LIN {X 0,Y 171.621,Z 603.214,A -85,B 0,C 180,E1 -26145.354,E2 -26145.354} C_VEL
LIN {X 0,Y 176.916,Z 615.978,A -85,B 0,C 180,E1 -26149,E2 -26149} C_VEL
LIN {X 0,Y 181.976,Z 626.134,A -85,B 0,C 180,E1 -26152.338,E2 -26152.338} C_VEL
LIN {X 0,Y 187.873,Z 635.706,A -85,B 0,C 180,E1 -26155.867,E2 -26155.867} C_VEL
LIN {X 0,Y 193.607,Z 643.258,A -85,B 0,C 180,E1 -26158.912,E2 -26158.912} C_VEL
LIN {X 0,Y 201.714,Z 651.879,A -85,B 0,C 180,E1 -26162.725,E2 -26162.725} C_VEL
LIN {X 0,Y 211.086,Z 659.54,A -85,B 0,C 180,E1 -26166.451,E2 -26166.451} C_VEL
LIN {X 0,Y 220.948,Z 665.783,A -85,B 0,C 180,E1 -26169.763,E2 -26169.763} C_VEL
LIN {X 0,Y 234.366,Z 672.498,A -85,B 0,C 180,E1 -26173.645,E2 -26173.645} C_VEL
LIN {X 0,Y 246.298,Z 677.555,A -85,B 0,C 180,E1 -26176.805,E2 -26176.805} C_VEL
LIN {X 0,Y 253.834,Z 680.558,A -85,B 0,C 180,E1 -26178.825,E2 -26178.825} C_VEL
LIN {X 0,Y 260.206,Z 683.111,A -85,B 0,C 180,E1 -26180.674,E2 -26180.674} C_VEL
LIN {X 0,Y 265.463,Z 685.211,A -85,B 0,C 180,E1 -26182.393,E2 -26182.393} C_VEL
LIN {X 0,Y 269.417,Z 686.886,A -85,B 0,C 180,E1 -26184.011,E2 -26184.011} C_VEL
LIN {X 0,Y 272.304,Z 688.198,A -85,B 0,C 180,E1 -26185.559,E2 -26185.559} C_VEL
LIN {X 0,Y 274.956,Z 689.105,A -85,B 0,C 180,E1 -26187.07,E2 -26187.07} C_VEL
LIN {X 0,Y 276.564,Z 689.664,A -85,B 0,C 180,E1 -26188.544,E2 -26188.544} C_VEL
LIN {X 0,Y 277.483,Z 689.842,A -85,B 0,C 180,E1 -26190,E2 -26190} C_VEL
LIN {X 0,Y 276.566,Z 689.663,A -85,B 0,C 180,E1 -26191.456,E2 -26191.456} C_VEL
LIN {X 0,Y 274.501,Z 688.974,A -85,B 0,C 180,E1 -26193.184,E2 -26193.184} C_VEL
LIN {X 0,Y 272.278,Z 688.199,A -85,B 0,C 180,E1 -26194.441,E2 -26194.441} C_VEL
LIN {X 0,Y 268.678,Z 686.595,A -85,B 0,C 180,E1 -26196.311,E2 -26196.311} C_VEL
LIN {X 0,Y 265.415,Z 685.213,A -85,B 0,C 180,E1 -26197.608,E2 -26197.608} C_VEL
LIN {X 0,Y 260.173,Z 683.112,A -85,B 0,C 180,E1 -26199.327,E2 -26199.327} C_VEL
LIN {X 0,Y 253.886,Z 680.557,A -85,B 0,C 180,E1 -26201.173,E2 -26201.173} C_VEL
LIN {X 0,Y 245.609,Z 677.259,A -85,B 0,C 180,E1 -26203.385,E2 -26203.385} C_VEL
LIN {X 0,Y 234.359,Z 672.513,A -85,B 0,C 180,E1 -26206.349,E2 -26206.349} C_VEL
LIN {X 0,Y 220.948,Z 665.784,A -85,B 0,C 180,E1 -26210.237,E2 -26210.237} C_VEL
LIN {X 0,Y 211.166,Z 659.537,A -85,B 0,C 180,E1 -26213.539,E2 -26213.539} C_VEL
LIN {X 0,Y 201.751,Z 651.903,A -85,B 0,C 180,E1 -26217.262,E2 -26217.262} C_VEL
LIN {X 0,Y 192.273,Z 641.586,A -85,B 0,C 180,E1 -26221.782,E2 -26221.782} C_VEL
LIN {X 0,Y 185.61,Z 632.244,A -85,B 0,C 180,E1 -26225.461,E2 -26225.461} C_VEL
LIN {X 0,Y 180.259,Z 622.941,A -85,B 0,C 180,E1 -26228.767,E2 -26228.767} C_VEL
LIN {X 0,Y 175.258,Z 612.247,A -85,B 0,C 180,E1 -26232.116,E2 -26232.116} C_VEL
LIN {X 0,Y 170.985,Z 601.587,A -85,B 0,C 180,E1 -26235.058,E2 -26235.058} C_VEL
LIN {X 0,Y 167.177,Z 590.937,A -85,B 0,C 180,E1 -26237.634,E2 -26237.634} C_VEL
LIN {X 0,Y 160.92,Z 572.907,A -85,B 0,C 180,E1 -26241.531,E2 -26241.531} C_VEL
LIN {X 0,Y 157.524,Z 564.607,A -85,B 0,C 180,E1 -26243.75,E2 -26243.75} C_VEL
LIN {X 0,Y 153.292,Z 555.729,A -85,B 0,C 180,E1 -26246.722,E2 -26246.722} C_VEL
LIN {X 0,Y 148.61,Z 547.106,A -85,B 0,C 180,E1 -26250.427,E2 -26250.427} C_VEL
LIN {X 0,Y 144.239,Z 539.962,A -85,B 0,C 180,E1 -26254.48,E2 -26254.48} C_VEL
LIN {X 0,Y 141.462,Z 535.851,A -85,B 0,C 180,E1 -26257.504,E2 -26257.504} C_VEL
LIN {X 0,Y 138.867,Z 531.989,A -85,B 0,C 180,E1 -26260.874,E2 -26260.874} C_VEL
LIN {X 0,Y 136.38,Z 528.521,A -85,B 0,C 180,E1 -26264.882,E2 -26264.882} C_VEL
LIN {X 0,Y 135.759,Z 527.362,A -85,B 0,C 180,E1 -26266.152,E2 -26266.152} C_VEL
LIN {X 0,Y 133.331,Z 524.419,A -85,B 0,C 180,E1 -26272.623,E2 -26272.623} C_VEL
LIN {X 0,Y 132.769,Z 522.602,A -85,B 0,C 180,E1 -26276.211,E2 -26276.211} C_VEL
LIN {X 0,Y 132.584,Z 521.985,A -85,B 0,C 180,E1 -26280.005,E2 -26280.005} C_VEL
LIN {X 0,Y 132.854,Z 522.928,A -85,B 0,C 180,E1 -26284.176,E2 -26284.176} C_VEL
LIN {X 0,Y 135.306,Z 527.03,A -85,B 0,C 180,E1 -26292.567,E2 -26292.567} C_VEL
LIN {X 0,Y 136.125,Z 527.942,A -85,B 0,C 180,E1 -26294.2,E2 -26294.2} C_VEL
LIN {X 0,Y 138.548,Z 531.658,A -85,B 0,C 180,E1 -26298.297,E2 -26298.297} C_VEL
LIN {X 0,Y 139.546,Z 533.014,A -85,B 0,C 180,E1 -26299.687,E2 -26299.687} C_VEL
LIN {X 0,Y 142.466,Z 537.271,A -85,B 0,C 180,E1 -26303.248,E2 -26303.248} C_VEL
LIN {X 0,Y 145.553,Z 542.106,A -85,B 0,C 180,E1 -26306.436,E2 -26306.436} C_VEL
LIN {X 0,Y 147.873,Z 546.115,A -85,B 0,C 180,E1 -26308.575,E2 -26308.575} C_VEL
LIN {X 0,Y 151.392,Z 554.209,A -85,B 0,C 180,E1 -26311.634,E2 -26311.634} C_VEL
LIN {X 0,Y 155.275,Z 564.625,A -85,B 0,C 180,E1 -26314.706,E2 -26314.706} C_VEL
LIN {X 0,Y 156.576,Z 568.776,A -85,B 0,C 180,E1 -26315.702,E2 -26315.702} C_VEL
LIN {X 0,Y 154.221,Z 595.964,A -85,B 0,C 180,E1 -26316.734,E2 -26316.734} C_VEL
LIN {X 0,Y 152.545,Z 606.818,A -85,B 0,C 180,E1 -26317.392,E2 -26317.392} C_VEL
LIN {X 0,Y 150.304,Z 616.608,A -85,B 0,C 180,E1 -26318.175,E2 -26318.175} C_VEL
LIN {X 0,Y 147.443,Z 626.404,A -85,B 0,C 180,E1 -26319.235,E2 -26319.235} C_VEL
LIN {X 0,Y 144.352,Z 635.168,A -85,B 0,C 180,E1 -26320.473,E2 -26320.473} C_VEL
LIN {X 0,Y 140.704,Z 643.886,A -85,B 0,C 180,E1 -26322.014,E2 -26322.014} C_VEL
LIN {X 0,Y 136.653,Z 652.394,A -85,B 0,C 180,E1 -26323.945,E2 -26323.945} C_VEL
LIN {X 0,Y 132.202,Z 660.561,A -85,B 0,C 180,E1 -26326.284,E2 -26326.284} C_VEL
LIN {X 0,Y 128.058,Z 667.504,A -85,B 0,C 180,E1 -26328.809,E2 -26328.809} C_VEL
LIN {X 0,Y 124.167,Z 673.491,A -85,B 0,C 180,E1 -26331.493,E2 -26331.493} C_VEL
LIN {X 0,Y 119.57,Z 680.174,A -85,B 0,C 180,E1 -26335.382,E2 -26335.382} C_VEL
LIN {X 0,Y 116.001,Z 685.08,A -85,B 0,C 180,E1 -26339.004,E2 -26339.004} C_VEL
LIN {X 0,Y 111.98,Z 690.174,A -85,B 0,C 180,E1 -26343.939,E2 -26343.939} C_VEL
LIN {X 0,Y 108.812,Z 694.141,A -85,B 0,C 180,E1 -26349.192,E2 -26349.192} C_VEL
LIN {X 0,Y 106.71,Z 697.085,A -85,B 0,C 180,E1 -26354.726,E2 -26354.726} C_VEL
LIN {X 0,Y 105.784,Z 698.592,A -85,B 0,C 180,E1 -26358.503,E2 -26358.503} C_VEL
LIN {X 0,Y 105.043,Z 700.131,A -85,B 0,C 180,E1 -26366.164,E2 -26366.164} C_VEL
LIN {X 0,Y 105.176,Z 700.418,A -85,B 0,C 180,E1 -26370,E2 -26370} C_VEL
LIN {X 0,Y 105.231,Z 699.528,A -85,B 0,C 180,E1 -26377.676,E2 -26377.676} C_VEL
LIN {X 0,Y 105.787,Z 698.592,A -85,B 0,C 180,E1 -26381.496,E2 -26381.496} C_VEL
LIN {X 0,Y 107.993,Z 695.232,A -85,B 0,C 180,E1 -26388.989,E2 -26388.989} C_VEL
LIN {X 0,Y 110.82,Z 691.602,A -85,B 0,C 180,E1 -26394.344,E2 -26394.344} C_VEL
LIN {X 0,Y 114.515,Z 686.868,A -85,B 0,C 180,E1 -26399.404,E2 -26399.404} C_VEL
LIN {X 0,Y 118.575,Z 681.494,A -85,B 0,C 180,E1 -26403.708,E2 -26403.708} C_VEL
LIN {X 0,Y 122.393,Z 676.116,A -85,B 0,C 180,E1 -26407.079,E2 -26407.079} C_VEL
LIN {X 0,Y 126.09,Z 670.624,A -85,B 0,C 180,E1 -26409.865,E2 -26409.865} C_VEL
LIN {X 0,Y 131.154,Z 662.411,A -85,B 0,C 180,E1 -26413.095,E2 -26413.095} C_VEL
LIN {X 0,Y 135.524,Z 654.59,A -85,B 0,C 180,E1 -26415.483,E2 -26415.483} C_VEL
LIN {X 0,Y 139.562,Z 646.512,A -85,B 0,C 180,E1 -26417.432,E2 -26417.432} C_VEL
LIN {X 0,Y 143.733,Z 636.756,A -85,B 0,C 180,E1 -26419.278,E2 -26419.278} C_VEL
LIN {X 0,Y 146.784,Z 628.37,A -85,B 0,C 180,E1 -26420.539,E2 -26420.539} C_VEL
LIN {X 0,Y 149.931,Z 617.868,A -85,B 0,C 180,E1 -26421.734,E2 -26421.734} C_VEL
LIN {X 0,Y 152.26,Z 608.189,A -85,B 0,C 180,E1 -26422.532,E2 -26422.532} C_VEL
LIN {X 0,Y 154.059,Z 597.555,A -85,B 0,C 180,E1 -26423.167,E2 -26423.167} C_VEL
LIN {X 0,Y 155.953,Z 576.912,A -85,B 0,C 180,E1 -26423.989,E2 -26423.989} C_VEL
LIN {X 0,Y 156.52,Z 568.606,A -85,B 0,C 180,E1 -26424.339,E2 -26424.339} C_VEL
LIN {X 0,Y 153.874,Z 560.714,A -85,B 0,C 180,E1 -26426.368,E2 -26426.368} C_VEL
LIN {X 0,Y 149.72,Z 550.16,A -85,B 0,C 180,E1 -26429.786,E2 -26429.786} C_VEL
LIN {X 0,Y 147.011,Z 544.436,A -85,B 0,C 180,E1 -26432.214,E2 -26432.214} C_VEL
LIN {X 0,Y 143.831,Z 539.389,A -85,B 0,C 180,E1 -26435.281,E2 -26435.281} C_VEL
LIN {X 0,Y 142.084,Z 536.551,A -85,B 0,C 180,E1 -26437.2,E2 -26437.2} C_VEL
LIN {X 0,Y 140.892,Z 535.032,A -85,B 0,C 180,E1 -26438.576,E2 -26438.576} C_VEL
LIN {X 0,Y 138.995,Z 533.903,A -85,B 0,C 180,E1 -26440.815,E2 -26440.815} C_VEL
LIN {X 0,Y 133.719,Z 533.482,A -85,B 0,C 180,E1 -26448.992,E2 -26448.992} C_VEL
LIN {X 0,Y 133.382,Z 533.176,A -85,B 0,C 180,E1 -26449.838,E2 -26449.838} C_VEL
LIN {X 0,Y 131.799,Z 529.387,A -85,B 0,C 180,E1 -26457.703,E2 -26457.703} C_VEL
LIN {X 0,Y 131.717,Z 529.047,A -85,B 0,C 180,E1 -26459.995,E2 -26459.995} C_VEL
LIN {X 0,Y 131.926,Z 529.956,A -85,B 0,C 180,E1 -26464.196,E2 -26464.196} C_VEL
LIN {X 0,Y 134.158,Z 533.971,A -85,B 0,C 180,E1 -26472.428,E2 -26472.428} C_VEL
LIN {X 0,Y 134.782,Z 534.696,A -85,B 0,C 180,E1 -26473.758,E2 -26473.758} C_VEL
LIN {X 0,Y 137.254,Z 538.568,A -85,B 0,C 180,E1 -26478.18,E2 -26478.18} C_VEL
LIN {X 0,Y 140.569,Z 543.731,A -85,B 0,C 180,E1 -26482.647,E2 -26482.647} C_VEL
LIN {X 0,Y 143.405,Z 548.348,A -85,B 0,C 180,E1 -26485.777,E2 -26485.777} C_VEL
LIN {X 0,Y 147.758,Z 556.106,A -85,B 0,C 180,E1 -26489.858,E2 -26489.858} C_VEL
LIN {X 0,Y 152.402,Z 565.552,A -85,B 0,C 180,E1 -26493.594,E2 -26493.594} C_VEL
LIN {X 0,Y 156.256,Z 574.926,A -85,B 0,C 180,E1 -26496.401,E2 -26496.401} C_VEL
LIN {X 0,Y 160.04,Z 586.179,A -85,B 0,C 180,E1 -26499.036,E2 -26499.036} C_VEL
LIN {X 0,Y 163.433,Z 597.185,A -85,B 0,C 180,E1 -26501.588,E2 -26501.588} C_VEL
LIN {X 0,Y 166.658,Z 607.047,A -85,B 0,C 180,E1 -26504.202,E2 -26504.202} C_VEL
LIN {X 0,Y 170.411,Z 617.155,A -85,B 0,C 180,E1 -26507.266,E2 -26507.266} C_VEL
LIN {X 0,Y 174.824,Z 627.17,A -85,B 0,C 180,E1 -26510.695,E2 -26510.695} C_VEL
LIN {X 0,Y 179.681,Z 635.973,A -85,B 0,C 180,E1 -26514.077,E2 -26514.077} C_VEL
LIN {X 0,Y 184.854,Z 643.572,A -85,B 0,C 180,E1 -26517.273,E2 -26517.273} C_VEL
LIN {X 0,Y 192.277,Z 652.277,A -85,B 0,C 180,E1 -26521.302,E2 -26521.302} C_VEL
LIN {X 0,Y 200.736,Z 659.845,A -85,B 0,C 180,E1 -26525.157,E2 -26525.157} C_VEL
LIN {X 0,Y 210.803,Z 666.663,A -85,B 0,C 180,E1 -26528.976,E2 -26528.976} C_VEL
LIN {X 0,Y 221.28,Z 672.126,A -85,B 0,C 180,E1 -26532.318,E2 -26532.318} C_VEL
LIN {X 0,Y 235.082,Z 677.867,A -85,B 0,C 180,E1 -26536.163,E2 -26536.163} C_VEL
LIN {X 0,Y 246.752,Z 682.108,A -85,B 0,C 180,E1 -26539.288,E2 -26539.288} C_VEL
LIN {X 0,Y 255.57,Z 685.165,A -85,B 0,C 180,E1 -26541.858,E2 -26541.858} C_VEL
LIN {X 0,Y 261.463,Z 687.257,A -85,B 0,C 180,E1 -26543.981,E2 -26543.981} C_VEL
LIN {X 0,Y 264.432,Z 688.418,A -85,B 0,C 180,E1 -26545.427,E2 -26545.427} C_VEL
LIN {X 0,Y 267.399,Z 689.359,A -85,B 0,C 180,E1 -26547.069,E2 -26547.069} C_VEL
LIN {X 0,Y 269.242,Z 689.867,A -85,B 0,C 180,E1 -26548.504,E2 -26548.504} C_VEL
LIN {X 0,Y 270.315,Z 690.041,A -85,B 0,C 180,E1 -26550,E2 -26550} C_VEL
LIN {X 0,Y 269.24,Z 689.867,A -85,B 0,C 180,E1 -26551.496,E2 -26551.496} C_VEL
LIN {X 0,Y 267.239,Z 689.317,A -85,B 0,C 180,E1 -26553.015,E2 -26553.015} C_VEL
LIN {X 0,Y 264.41,Z 688.418,A -85,B 0,C 180,E1 -26554.574,E2 -26554.574} C_VEL
LIN {X 0,Y 261.016,Z 687.117,A -85,B 0,C 180,E1 -26556.183,E2 -26556.183} C_VEL
LIN {X 0,Y 255.564,Z 685.178,A -85,B 0,C 180,E1 -26558.132,E2 -26558.132} C_VEL
LIN {X 0,Y 249.679,Z 683.135,A -85,B 0,C 180,E1 -26559.893,E2 -26559.893} C_VEL
LIN {X 0,Y 243.252,Z 680.857,A -85,B 0,C 180,E1 -26561.668,E2 -26561.668} C_VEL
LIN {X 0,Y 232.346,Z 676.846,A -85,B 0,C 180,E1 -26564.562,E2 -26564.562} C_VEL
LIN {X 0,Y 217.434,Z 670.286,A -85,B 0,C 180,E1 -26568.858,E2 -26568.858} C_VEL
LIN {X 0,Y 205.884,Z 663.53,A -85,B 0,C 180,E1 -26572.839,E2 -26572.839} C_VEL
LIN {X 0,Y 195.479,Z 655.394,A -85,B 0,C 180,E1 -26577.158,E2 -26577.158} C_VEL
LIN {X 0,Y 188.213,Z 647.777,A -85,B 0,C 180,E1 -26580.821,E2 -26580.821} C_VEL
LIN {X 0,Y 181.58,Z 639.028,A -85,B 0,C 180,E1 -26584.674,E2 -26584.674} C_VEL
LIN {X 0,Y 176.615,Z 630.661,A -85,B 0,C 180,E1 -26588.007,E2 -26588.007} C_VEL
LIN {X 0,Y 172.513,Z 622.049,A -85,B 0,C 180,E1 -26591.095,E2 -26591.095} C_VEL
LIN {X 0,Y 168.754,Z 612.855,A -85,B 0,C 180,E1 -26594.083,E2 -26594.083} C_VEL
LIN {X 0,Y 164.892,Z 601.852,A -85,B 0,C 180,E1 -26597.218,E2 -26597.218} C_VEL
LIN {X 0,Y 161.241,Z 590.184,A -85,B 0,C 180,E1 -26600.098,E2 -26600.098} C_VEL
LIN {X 0,Y 156.857,Z 576.56,A -85,B 0,C 180,E1 -26603.178,E2 -26603.178} C_VEL
LIN {X 0,Y 152.863,Z 566.622,A -85,B 0,C 180,E1 -26606.056,E2 -26606.056} C_VEL
LIN {X 0,Y 148.504,Z 557.612,A -85,B 0,C 180,E1 -26609.499,E2 -26609.499} C_VEL
LIN {X 0,Y 144.243,Z 549.708,A -85,B 0,C 180,E1 -26613.387,E2 -26613.387} C_VEL
LIN {X 0,Y 141.473,Z 545.217,A -85,B 0,C 180,E1 -26616.297,E2 -26616.297} C_VEL
LIN {X 0,Y 139.46,Z 542.029,A -85,B 0,C 180,E1 -26618.719,E2 -26618.719} C_VEL
LIN {X 0,Y 137.255,Z 538.56,A -85,B 0,C 180,E1 -26621.819,E2 -26621.819} C_VEL
LIN {X 0,Y 134.781,Z 534.7,A -85,B 0,C 180,E1 -26626.242,E2 -26626.242} C_VEL
LIN {X 0,Y 134.159,Z 533.961,A -85,B 0,C 180,E1 -26627.572,E2 -26627.572} C_VEL
LIN {X 0,Y 131.822,Z 529.519,A -85,B 0,C 180,E1 -26636.949,E2 -26636.949} C_VEL
LIN {X 0,Y 131.718,Z 529.04,A -85,B 0,C 180,E1 -26640.005,E2 -26640.005} C_VEL
LIN {X 0,Y 131.94,Z 529.991,A -85,B 0,C 180,E1 -26643.918,E2 -26643.918} C_VEL
LIN {X 0,Y 134.319,Z 534.061,A -85,B 0,C 180,E1 -26652.373,E2 -26652.373} C_VEL
LIN {X 0,Y 134.87,Z 534.887,A -85,B 0,C 180,E1 -26653.566,E2 -26653.566} C_VEL
LIN {X 0,Y 137.881,Z 539.509,A -85,B 0,C 180,E1 -26658.726,E2 -26658.726} C_VEL
LIN {X 0,Y 140.659,Z 543.824,A -85,B 0,C 180,E1 -26662.359,E2 -26662.359} C_VEL
LIN {X 0,Y 144.231,Z 549.666,A -85,B 0,C 180,E1 -26666.21,E2 -26666.21} C_VEL
LIN {X 0,Y 146.772,Z 555.356,A -85,B 0,C 180,E1 -26668.712,E2 -26668.712} C_VEL
LIN {X 0,Y 150.791,Z 566.153,A -85,B 0,C 180,E1 -26672.316,E2 -26672.316} C_VEL
LIN {X 0,Y 152.326,Z 571.077,A -85,B 0,C 180,E1 -26673.622,E2 -26673.622} C_VEL
LIN {X 0,Y 150.034,Z 596.193,A -85,B 0,C 180,E1 -26674.584,E2 -26674.584} C_VEL
LIN {X 0,Y 148.095,Z 608.002,A -85,B 0,C 180,E1 -26675.314,E2 -26675.314} C_VEL
LIN {X 0,Y 144.712,Z 621.282,A -85,B 0,C 180,E1 -26676.452,E2 -26676.452} C_VEL
LIN {X 0,Y 140.507,Z 633.383,A -85,B 0,C 180,E1 -26678.021,E2 -26678.021} C_VEL
LIN {X 0,Y 136.691,Z 642.379,A -85,B 0,C 180,E1 -26679.536,E2 -26679.536} C_VEL
LIN {X 0,Y 132.434,Z 651.101,A -85,B 0,C 180,E1 -26681.446,E2 -26681.446} C_VEL
LIN {X 0,Y 128.308,Z 658.516,A -85,B 0,C 180,E1 -26683.469,E2 -26683.469} C_VEL
LIN {X 0,Y 122.797,Z 667.308,A -85,B 0,C 180,E1 -26686.624,E2 -26686.624} C_VEL
LIN {X 0,Y 118.669,Z 673.294,A -85,B 0,C 180,E1 -26689.349,E2 -26689.349} C_VEL
LIN {X 0,Y 114.952,Z 678.499,A -85,B 0,C 180,E1 -26692.311,E2 -26692.311} C_VEL
LIN {X 0,Y 109.964,Z 684.884,A -85,B 0,C 180,E1 -26697.095,E2 -26697.095} C_VEL
LIN {X 0,Y 105.619,Z 689.977,A -85,B 0,C 180,E1 -26702.239,E2 -26702.239} C_VEL
LIN {X 0,Y 102.189,Z 693.944,A -85,B 0,C 180,E1 -26707.774,E2 -26707.774} C_VEL
LIN {X 0,Y 99.835,Z 696.887,A -85,B 0,C 180,E1 -26713.645,E2 -26713.645} C_VEL
LIN {X 0,Y 98.804,Z 698.395,A -85,B 0,C 180,E1 -26717.679,E2 -26717.679} C_VEL
LIN {X 0,Y 97.949,Z 699.935,A -85,B 0,C 180,E1 -26725.885,E2 -26725.885} C_VEL
LIN {X 0,Y 98.083,Z 700.222,A -85,B 0,C 180,E1 -26730,E2 -26730} C_VEL
LIN {X 0,Y 98.188,Z 699.331,A -85,B 0,C 180,E1 -26738.23,E2 -26738.23} C_VEL
LIN {X 0,Y 98.806,Z 698.395,A -85,B 0,C 180,E1 -26742.321,E2 -26742.321} C_VEL
LIN {X 0,Y 101.264,Z 695.034,A -85,B 0,C 180,E1 -26750.305,E2 -26750.305} C_VEL
LIN {X 0,Y 104.361,Z 691.405,A -85,B 0,C 180,E1 -26755.959,E2 -26755.959} C_VEL
LIN {X 0,Y 108.374,Z 686.672,A -85,B 0,C 180,E1 -26761.251,E2 -26761.251} C_VEL
LIN {X 0,Y 113.448,Z 680.404,A -85,B 0,C 180,E1 -26766.349,E2 -26766.349} C_VEL
LIN {X 0,Y 118.688,Z 673.295,A -85,B 0,C 180,E1 -26770.643,E2 -26770.643} C_VEL
LIN {X 0,Y 124.948,Z 664.064,A -85,B 0,C 180,E1 -26774.675,E2 -26774.675} C_VEL
LIN {X 0,Y 130.628,Z 654.393,A -85,B 0,C 180,E1 -26777.712,E2 -26777.712} C_VEL
LIN {X 0,Y 134.865,Z 646.316,A -85,B 0,C 180,E1 -26779.651,E2 -26779.651} C_VEL
LIN {X 0,Y 139.205,Z 636.56,A -85,B 0,C 180,E1 -26781.493,E2 -26781.493} C_VEL
LIN {X 0,Y 142.377,Z 628.174,A -85,B 0,C 180,E1 -26782.745,E2 -26782.745} C_VEL
LIN {X 0,Y 145.646,Z 617.672,A -85,B 0,C 180,E1 -26783.925,E2 -26783.925} C_VEL
LIN {X 0,Y 148.205,Z 607.314,A -85,B 0,C 180,E1 -26784.743,E2 -26784.743} C_VEL
LIN {X 0,Y 149.975,Z 596.932,A -85,B 0,C 180,E1 -26785.351,E2 -26785.351} C_VEL
LIN {X 0,Y 151.985,Z 575.616,A -85,B 0,C 180,E1 -26786.192,E2 -26786.192} C_VEL
LIN {X 0,Y 152.233,Z 570.793,A -85,B 0,C 180,E1 -26786.453,E2 -26786.453} C_VEL
LIN {X 0,Y 150.06,Z 564.182,A -85,B 0,C 180,E1 -26788.299,E2 -26788.299} C_VEL
LIN {X 0,Y 146.442,Z 554.498,A -85,B 0,C 180,E1 -26791.609,E2 -26791.609} C_VEL
LIN {X 0,Y 144.15,Z 549.512,A -85,B 0,C 180,E1 -26793.872,E2 -26793.872} C_VEL
LIN {X 0,Y 140.041,Z 542.737,A -85,B 0,C 180,E1 -26798.404,E2 -26798.404} C_VEL
LIN {X 0,Y 137.085,Z 538.343,A -85,B 0,C 180,E1 -26802.466,E2 -26802.466} C_VEL
LIN {X 0,Y 134.697,Z 534.461,A -85,B 0,C 180,E1 -26806.834,E2 -26806.834} C_VEL
LIN {X 0,Y 133.382,Z 533.176,A -85,B 0,C 180,E1 -26809.838,E2 -26809.838} C_VEL
LIN {X 0,Y 132.512,Z 532.627,A -85,B 0,C 180,E1 -26812.365,E2 -26812.365} C_VEL
LIN {X 0,Y 131.792,Z 532.955,A -85,B 0,C 180,E1 -26814.933,E2 -26814.933} C_VEL
LIN {X 0,Y 130.969,Z 535.132,A -85,B 0,C 180,E1 -26820.102,E2 -26820.102} C_VEL
LIN {X 0,Y 130.986,Z 536.834,A -85,B 0,C 180,E1 -26823.563,E2 -26823.563} C_VEL
LIN {X 0,Y 133.157,Z 540.966,A -85,B 0,C 180,E1 -26832.183,E2 -26832.183} C_VEL
LIN {X 0,Y 136.274,Z 546.089,A -85,B 0,C 180,E1 -26838.168,E2 -26838.168} C_VEL
LIN {X 0,Y 138.864,Z 550.396,A -85,B 0,C 180,E1 -26841.815,E2 -26841.815} C_VEL
LIN {X 0,Y 141.09,Z 554.185,A -85,B 0,C 180,E1 -26844.455,E2 -26844.455} C_VEL
LIN {X 0,Y 145.036,Z 561.671,A -85,B 0,C 180,E1 -26848.487,E2 -26848.487} C_VEL
LIN {X 0,Y 149.247,Z 570.719,A -85,B 0,C 180,E1 -26852.172,E2 -26852.172} C_VEL
LIN {X 0,Y 152.826,Z 579.943,A -85,B 0,C 180,E1 -26855.011,E2 -26855.011} C_VEL
LIN {X 0,Y 155.977,Z 590.349,A -85,B 0,C 180,E1 -26857.561,E2 -26857.561} C_VEL
LIN {X 0,Y 158.362,Z 599.183,A -85,B 0,C 180,E1 -26859.737,E2 -26859.737} C_VEL
LIN {X 0,Y 161.065,Z 608.7,A -85,B 0,C 180,E1 -26862.383,E2 -26862.383} C_VEL
LIN {X 0,Y 163.883,Z 617.554,A -85,B 0,C 180,E1 -26865.153,E2 -26865.153} C_VEL
LIN {X 0,Y 167.126,Z 626.218,A -85,B 0,C 180,E1 -26868.185,E2 -26868.185} C_VEL
LIN {X 0,Y 170.873,Z 634.482,A -85,B 0,C 180,E1 -26871.389,E2 -26871.389} C_VEL
LIN {X 0,Y 176.446,Z 644.006,A -85,B 0,C 180,E1 -26875.553,E2 -26875.553} C_VEL
LIN {X 0,Y 183.092,Z 652.655,A -85,B 0,C 180,E1 -26879.749,E2 -26879.749} C_VEL
LIN {X 0,Y 190.671,Z 660.146,A -85,B 0,C 180,E1 -26883.749,E2 -26883.749} C_VEL
LIN {X 0,Y 198.336,Z 665.908,A -85,B 0,C 180,E1 -26887.108,E2 -26887.108} C_VEL
LIN {X 0,Y 208.351,Z 671.711,A -85,B 0,C 180,E1 -26890.808,E2 -26890.808} C_VEL
LIN {X 0,Y 219.133,Z 676.52,A -85,B 0,C 180,E1 -26894.173,E2 -26894.173} C_VEL
LIN {X 0,Y 232.109,Z 681.172,A -85,B 0,C 180,E1 -26897.763,E2 -26897.763} C_VEL
LIN {X 0,Y 242.25,Z 684.363,A -85,B 0,C 180,E1 -26900.515,E2 -26900.515} C_VEL
LIN {X 0,Y 248.219,Z 686.173,A -85,B 0,C 180,E1 -26902.274,E2 -26902.274} C_VEL
LIN {X 0,Y 254.236,Z 687.958,A -85,B 0,C 180,E1 -26904.334,E2 -26904.334} C_VEL
LIN {X 0,Y 256.368,Z 688.643,A -85,B 0,C 180,E1 -26905.283,E2 -26905.283} C_VEL
LIN {X 0,Y 260.299,Z 689.748,A -85,B 0,C 180,E1 -26907.356,E2 -26907.356} C_VEL
LIN {X 0,Y 261.821,Z 690.072,A -85,B 0,C 180,E1 -26908.462,E2 -26908.462} C_VEL
LIN {X 0,Y 263.123,Z 690.239,A -85,B 0,C 180,E1 -26910,E2 -26910} C_VEL
LIN {X 0,Y 261.817,Z 690.071,A -85,B 0,C 180,E1 -26911.538,E2 -26911.538} C_VEL
LIN {X 0,Y 259.449,Z 689.531,A -85,B 0,C 180,E1 -26913.106,E2 -26913.106} C_VEL
LIN {X 0,Y 256.345,Z 688.643,A -85,B 0,C 180,E1 -26914.718,E2 -26914.718} C_VEL
LIN {X 0,Y 254.232,Z 687.965,A -85,B 0,C 180,E1 -26915.658,E2 -26915.658} C_VEL
LIN {X 0,Y 248.218,Z 686.176,A -85,B 0,C 180,E1 -26917.724,E2 -26917.724} C_VEL
LIN {X 0,Y 239.977,Z 683.679,A -85,B 0,C 180,E1 -26920.12,E2 -26920.12} C_VEL
LIN {X 0,Y 230.5,Z 680.631,A -85,B 0,C 180,E1 -26922.676,E2 -26922.676} C_VEL
LIN {X 0,Y 214.81,Z 674.704,A -85,B 0,C 180,E1 -26927.125,E2 -26927.125} C_VEL
LIN {X 0,Y 203.242,Z 668.921,A -85,B 0,C 180,E1 -26931,E2 -26931} C_VEL
LIN {X 0,Y 193.666,Z 662.535,A -85,B 0,C 180,E1 -26934.884,E2 -26934.884} C_VEL
LIN {X 0,Y 186.106,Z 655.804,A -85,B 0,C 180,E1 -26938.606,E2 -26938.606} C_VEL
LIN {X 0,Y 179.276,Z 647.971,A -85,B 0,C 180,E1 -26942.568,E2 -26942.568} C_VEL
LIN {X 0,Y 174.048,Z 640.217,A -85,B 0,C 180,E1 -26946.146,E2 -26946.146} C_VEL
LIN {X 0,Y 169.699,Z 632.112,A -85,B 0,C 180,E1 -26949.557,E2 -26949.557} C_VEL
LIN {X 0,Y 165.816,Z 622.857,A -85,B 0,C 180,E1 -26953.025,E2 -26953.025} C_VEL
LIN {X 0,Y 162.519,Z 613.253,A -85,B 0,C 180,E1 -26956.225,E2 -26956.225} C_VEL
LIN {X 0,Y 159.259,Z 602.507,A -85,B 0,C 180,E1 -26959.396,E2 -26959.396} C_VEL
LIN {X 0,Y 156.191,Z 591.08,A -85,B 0,C 180,E1 -26962.296,E2 -26962.296} C_VEL
LIN {X 0,Y 152.909,Z 580.112,A -85,B 0,C 180,E1 -26964.93,E2 -26964.93} C_VEL
LIN {X 0,Y 149.16,Z 570.549,A -85,B 0,C 180,E1 -26967.896,E2 -26967.896} C_VEL
LIN {X 0,Y 145.19,Z 562.04,A -85,B 0,C 180,E1 -26971.363,E2 -26971.363} C_VEL
LIN {X 0,Y 141.548,Z 554.977,A -85,B 0,C 180,E1 -26975.042,E2 -26975.042} C_VEL
LIN {X 0,Y 138.144,Z 549.065,A -85,B 0,C 180,E1 -26979.143,E2 -26979.143} C_VEL
LIN {X 0,Y 135.497,Z 544.882,A -85,B 0,C 180,E1 -26983.09,E2 -26983.09} C_VEL
LIN {X 0,Y 133.157,Z 540.966,A -85,B 0,C 180,E1 -26987.817,E2 -26987.817} C_VEL
LIN {X 0,Y 131.111,Z 537.419,A -85,B 0,C 180,E1 -26995.2,E2 -26995.2} C_VEL
LIN {X 0,Y 130.897,Z 536.44,A -85,B 0,C 180,E1 -26997.697,E2 -26997.697} C_VEL
LIN {X 0,Y 130.857,Z 536.195,A -85,B 0,C 180,E1 -27000.774,E2 -27000.774} C_VEL
LIN {X 0,Y 131.03,Z 537.046,A -85,B 0,C 180,E1 -27003.657,E2 -27003.657} C_VEL
LIN {X 0,Y 133.164,Z 540.952,A -85,B 0,C 180,E1 -27011.805,E2 -27011.805} C_VEL
LIN {X 0,Y 136.198,Z 545.92,A -85,B 0,C 180,E1 -27017.652,E2 -27017.652} C_VEL
LIN {X 0,Y 138.95,Z 550.524,A -85,B 0,C 180,E1 -27021.532,E2 -27021.532} C_VEL
LIN {X 0,Y 141.931,Z 555.68,A -85,B 0,C 180,E1 -27024.984,E2 -27024.984} C_VEL
LIN {X 0,Y 144.41,Z 561.744,A -85,B 0,C 180,E1 -27027.641,E2 -27027.641} C_VEL
LIN {X 0,Y 148.057,Z 572.635,A -85,B 0,C 180,E1 -27031.213,E2 -27031.213} C_VEL
LIN {X 0,Y 148.279,Z 573.652,A -85,B 0,C 180,E1 -27031.445,E2 -27031.445} C_VEL
LIN {X 0,Y 146.028,Z 596.711,A -85,B 0,C 180,E1 -27032.325,E2 -27032.325} C_VEL
LIN {X 0,Y 143.82,Z 609.218,A -85,B 0,C 180,E1 -27033.097,E2 -27033.097} C_VEL
LIN {X 0,Y 140.279,Z 622.078,A -85,B 0,C 180,E1 -27034.245,E2 -27034.245} C_VEL
LIN {X 0,Y 136.248,Z 633.187,A -85,B 0,C 180,E1 -27035.668,E2 -27035.668} C_VEL
LIN {X 0,Y 132.275,Z 642.182,A -85,B 0,C 180,E1 -27037.159,E2 -27037.159} C_VEL
LIN {X 0,Y 127.837,Z 650.904,A -85,B 0,C 180,E1 -27039.056,E2 -27039.056} C_VEL
LIN {X 0,Y 123.532,Z 658.32,A -85,B 0,C 180,E1 -27041.078,E2 -27041.078} C_VEL
LIN {X 0,Y 117.728,Z 667.111,A -85,B 0,C 180,E1 -27044.245,E2 -27044.245} C_VEL
LIN {X 0,Y 113.364,Z 673.098,A -85,B 0,C 180,E1 -27047.005,E2 -27047.005} C_VEL
LIN {X 0,Y 108.289,Z 679.596,A -85,B 0,C 180,E1 -27050.95,E2 -27050.95} C_VEL
LIN {X 0,Y 104.058,Z 684.687,A -85,B 0,C 180,E1 -27054.965,E2 -27054.965} C_VEL
LIN {X 0,Y 99.35,Z 689.779,A -85,B 0,C 180,E1 -27060.319,E2 -27060.319} C_VEL
LIN {X 0,Y 95.616,Z 693.746,A -85,B 0,C 180,E1 -27066.155,E2 -27066.155} C_VEL
LIN {X 0,Y 93.01,Z 696.69,A -85,B 0,C 180,E1 -27072.408,E2 -27072.408} C_VEL
LIN {X 0,Y 91.857,Z 698.198,A -85,B 0,C 180,E1 -27076.731,E2 -27076.731} C_VEL
LIN {X 0,Y 90.879,Z 699.739,A -85,B 0,C 180,E1 -27085.565,E2 -27085.565} C_VEL
LIN {X 0,Y 90.981,Z 700.026,A -85,B 0,C 180,E1 -27090,E2 -27090} C_VEL
LIN {X 0,Y 91.149,Z 699.134,A -85,B 0,C 180,E1 -27098.871,E2 -27098.871} C_VEL
LIN {X 0,Y 91.859,Z 698.198,A -85,B 0,C 180,E1 -27103.269,E2 -27103.269} C_VEL
LIN {X 0,Y 94.601,Z 694.837,A -85,B 0,C 180,E1 -27111.805,E2 -27111.805} C_VEL
LIN {X 0,Y 98.001,Z 691.208,A -85,B 0,C 180,E1 -27117.784,E2 -27117.784} C_VEL
LIN {X 0,Y 102.362,Z 686.475,A -85,B 0,C 180,E1 -27123.316,E2 -27123.316} C_VEL
LIN {X 0,Y 105.72,Z 682.688,A -85,B 0,C 180,E1 -27126.748,E2 -27126.748} C_VEL
LIN {X 0,Y 110.349,Z 677.033,A -85,B 0,C 180,E1 -27130.753,E2 -27130.753} C_VEL
LIN {X 0,Y 115.515,Z 670.231,A -85,B 0,C 180,E1 -27134.4,E2 -27134.4} C_VEL
LIN {X 0,Y 121.155,Z 662.018,A -85,B 0,C 180,E1 -27137.697,E2 -27137.697} C_VEL
LIN {X 0,Y 125.962,Z 654.197,A -85,B 0,C 180,E1 -27140.1,E2 -27140.1} C_VEL
LIN {X 0,Y 130.369,Z 646.119,A -85,B 0,C 180,E1 -27142.037,E2 -27142.037} C_VEL
LIN {X 0,Y 134.893,Z 636.364,A -85,B 0,C 180,E1 -27143.857,E2 -27143.857} C_VEL
LIN {X 0,Y 138.201,Z 627.978,A -85,B 0,C 180,E1 -27145.085,E2 -27145.085} C_VEL
LIN {X 0,Y 141.591,Z 617.476,A -85,B 0,C 180,E1 -27146.242,E2 -27146.242} C_VEL
LIN {X 0,Y 144.291,Z 606.704,A -85,B 0,C 180,E1 -27147.083,E2 -27147.083} C_VEL
LIN {X 0,Y 146.058,Z 596.62,A -85,B 0,C 180,E1 -27147.655,E2 -27147.655} C_VEL
LIN {X 0,Y 148.301,Z 573.653,A -85,B 0,C 180,E1 -27148.541,E2 -27148.541} C_VEL
LIN {X 0,Y 146.446,Z 567.698,A -85,B 0,C 180,E1 -27150.308,E2 -27150.308} C_VEL
LIN {X 0,Y 143.238,Z 558.686,A -85,B 0,C 180,E1 -27153.594,E2 -27153.594} C_VEL
LIN {X 0,Y 141.591,Z 555.062,A -85,B 0,C 180,E1 -27155.383,E2 -27155.383} C_VEL
LIN {X 0,Y 138.221,Z 549.136,A -85,B 0,C 180,E1 -27159.438,E2 -27159.438} C_VEL
LIN {X 0,Y 135.425,Z 544.757,A -85,B 0,C 180,E1 -27163.604,E2 -27163.604} C_VEL
LIN {X 0,Y 133.164,Z 540.956,A -85,B 0,C 180,E1 -27168.195,E2 -27168.195} C_VEL
LIN {X 0,Y 130.929,Z 536.476,A -85,B 0,C 180,E1 -27177.688,E2 -27177.688} C_VEL
LIN {X 0,Y 130.85,Z 536.104,A -85,B 0,C 180,E1 -27179.995,E2 -27179.995} C_VEL
LIN {X 0,Y 130.986,Z 536.834,A -85,B 0,C 180,E1 -27183.563,E2 -27183.563} C_VEL
LIN {X 0,Y 131.078,Z 538.295,A -85,B 0,C 180,E1 -27185.19,E2 -27185.19} C_VEL
LIN {X 0,Y 131.458,Z 546.478,A -85,B 0,C 180,E1 -27189.901,E2 -27189.901} C_VEL
LIN {X 0,Y 131.977,Z 547.819,A -85,B 0,C 180,E1 -27191.51,E2 -27191.51} C_VEL
LIN {X 0,Y 134.764,Z 552.764,A -85,B 0,C 180,E1 -27197.298,E2 -27197.298} C_VEL
LIN {X 0,Y 137.158,Z 557.016,A -85,B 0,C 180,E1 -27200.92,E2 -27200.92} C_VEL
LIN {X 0,Y 139.714,Z 561.676,A -85,B 0,C 180,E1 -27204.119,E2 -27204.119} C_VEL
LIN {X 0,Y 143.51,Z 569.641,A -85,B 0,C 180,E1 -27208.177,E2 -27208.177} C_VEL
LIN {X 0,Y 146.765,Z 577.39,A -85,B 0,C 180,E1 -27211.211,E2 -27211.211} C_VEL
LIN {X 0,Y 149.807,Z 586.034,A -85,B 0,C 180,E1 -27213.85,E2 -27213.85} C_VEL
LIN {X 0,Y 152.83,Z 598.455,A -85,B 0,C 180,E1 -27217.017,E2 -27217.017} C_VEL
LIN {X 0,Y 155.346,Z 609.108,A -85,B 0,C 180,E1 -27220.051,E2 -27220.051} C_VEL
LIN {X 0,Y 157.713,Z 618.028,A -85,B 0,C 180,E1 -27222.934,E2 -27222.934} C_VEL
LIN {X 0,Y 160.547,Z 627.138,A -85,B 0,C 180,E1 -27226.236,E2 -27226.236} C_VEL
LIN {X 0,Y 164.211,Z 636.496,A -85,B 0,C 180,E1 -27230.061,E2 -27230.061} C_VEL
LIN {X 0,Y 168.342,Z 644.366,A -85,B 0,C 180,E1 -27233.671,E2 -27233.671} C_VEL
LIN {X 0,Y 174.097,Z 652.807,A -85,B 0,C 180,E1 -27237.958,E2 -27237.958} C_VEL
LIN {X 0,Y 181.057,Z 660.437,A -85,B 0,C 180,E1 -27242.239,E2 -27242.239} C_VEL
LIN {X 0,Y 189.316,Z 667.107,A -85,B 0,C 180,E1 -27246.372,E2 -27246.372} C_VEL
LIN {X 0,Y 198.155,Z 672.483,A -85,B 0,C 180,E1 -27250.02,E2 -27250.02} C_VEL
LIN {X 0,Y 208.731,Z 677.329,A -85,B 0,C 180,E1 -27253.645,E2 -27253.645} C_VEL
LIN {X 0,Y 222.918,Z 682.217,A -85,B 0,C 180,E1 -27257.765,E2 -27257.765} C_VEL
LIN {X 0,Y 228.928,Z 683.991,A -85,B 0,C 180,E1 -27259.386,E2 -27259.386} C_VEL
LIN {X 0,Y 236.566,Z 686.005,A -85,B 0,C 180,E1 -27261.458,E2 -27261.458} C_VEL
LIN {X 0,Y 242.966,Z 687.615,A -85,B 0,C 180,E1 -27263.356,E2 -27263.356} C_VEL
LIN {X 0,Y 248.091,Z 688.874,A -85,B 0,C 180,E1 -27265.125,E2 -27265.125} C_VEL
LIN {X 0,Y 253.206,Z 690.072,A -85,B 0,C 180,E1 -27267.655,E2 -27267.655} C_VEL
LIN {X 0,Y 254.33,Z 690.277,A -85,B 0,C 180,E1 -27268.417,E2 -27268.417} C_VEL
LIN {X 0,Y 255.899,Z 690.439,A -85,B 0,C 180,E1 -27270,E2 -27270} C_VEL
LIN {X 0,Y 254.324,Z 690.277,A -85,B 0,C 180,E1 -27271.583,E2 -27271.583} C_VEL
LIN {X 0,Y 251.531,Z 689.748,A -85,B 0,C 180,E1 -27273.203,E2 -27273.203} C_VEL
LIN {X 0,Y 248.07,Z 688.874,A -85,B 0,C 180,E1 -27274.876,E2 -27274.876} C_VEL
LIN {X 0,Y 240.884,Z 687.129,A -85,B 0,C 180,E1 -27277.288,E2 -27277.288} C_VEL
LIN {X 0,Y 234.82,Z 685.533,A -85,B 0,C 180,E1 -27279.03,E2 -27279.03} C_VEL
LIN {X 0,Y 228.825,Z 683.946,A -85,B 0,C 180,E1 -27280.652,E2 -27280.652} C_VEL
LIN {X 0,Y 217.138,Z 680.417,A -85,B 0,C 180,E1 -27283.848,E2 -27283.848} C_VEL
LIN {X 0,Y 203.352,Z 675.034,A -85,B 0,C 180,E1 -27288.122,E2 -27288.122} C_VEL
LIN {X 0,Y 193.756,Z 669.986,A -85,B 0,C 180,E1 -27291.734,E2 -27291.734} C_VEL
LIN {X 0,Y 184.021,Z 663.092,A -85,B 0,C 180,E1 -27296.178,E2 -27296.178} C_VEL
LIN {X 0,Y 176.901,Z 656.128,A -85,B 0,C 180,E1 -27300.23,E2 -27300.23} C_VEL
LIN {X 0,Y 170.576,Z 648.064,A -85,B 0,C 180,E1 -27304.517,E2 -27304.517} C_VEL
LIN {X 0,Y 165.878,Z 639.955,A -85,B 0,C 180,E1 -27308.396,E2 -27308.396} C_VEL
LIN {X 0,Y 162.12,Z 631.327,A -85,B 0,C 180,E1 -27312.088,E2 -27312.088} C_VEL
LIN {X 0,Y 158.928,Z 622.166,A -85,B 0,C 180,E1 -27315.612,E2 -27315.612} C_VEL
LIN {X 0,Y 156.235,Z 612.579,A -85,B 0,C 180,E1 -27318.869,E2 -27318.869} C_VEL
LIN {X 0,Y 153.76,Z 602.382,A -85,B 0,C 180,E1 -27321.904,E2 -27321.904} C_VEL
LIN {X 0,Y 151.316,Z 591.592,A -85,B 0,C 180,E1 -27324.719,E2 -27324.719} C_VEL
LIN {X 0,Y 148.543,Z 582.164,A -85,B 0,C 180,E1 -27327.244,E2 -27327.244} C_VEL
LIN {X 0,Y 145.153,Z 573.427,A -85,B 0,C 180,E1 -27330.251,E2 -27330.251} C_VEL
LIN {X 0,Y 141.601,Z 565.559,A -85,B 0,C 180,E1 -27333.771,E2 -27333.771} C_VEL
LIN {X 0,Y 138.095,Z 558.582,A -85,B 0,C 180,E1 -27337.861,E2 -27337.861} C_VEL
LIN {X 0,Y 135.718,Z 554.473,A -85,B 0,C 180,E1 -27341.159,E2 -27341.159} C_VEL
LIN {X 0,Y 134.115,Z 551.634,A -85,B 0,C 180,E1 -27343.841,E2 -27343.841} C_VEL
LIN {X 0,Y 131.983,Z 547.826,A -85,B 0,C 180,E1 -27348.475,E2 -27348.475} C_VEL
LIN {X 0,Y 130.115,Z 544.039,A -85,B 0,C 180,E1 -27356.327,E2 -27356.327} C_VEL
LIN {X 0,Y 129.979,Z 543.251,A -85,B 0,C 180,E1 -27359.23,E2 -27359.23} C_VEL
LIN {X 0,Y 130.054,Z 543.611,A -85,B 0,C 180,E1 -27362.328,E2 -27362.328} C_VEL
LIN {X 0,Y 132.278,Z 548.331,A -85,B 0,C 180,E1 -27371.886,E2 -27371.886} C_VEL
LIN {X 0,Y 134.823,Z 552.841,A -85,B 0,C 180,E1 -27377.005,E2 -27377.005} C_VEL
LIN {X 0,Y 137.228,Z 557.096,A -85,B 0,C 180,E1 -27380.62,E2 -27380.62} C_VEL
LIN {X 0,Y 139.931,Z 562.171,A -85,B 0,C 180,E1 -27383.99,E2 -27383.99} C_VEL
LIN {X 0,Y 142.331,Z 569.087,A -85,B 0,C 180,E1 -27386.822,E2 -27386.822} C_VEL
LIN {X 0,Y 144.462,Z 575.847,A -85,B 0,C 180,E1 -27389.115,E2 -27389.115} C_VEL
LIN {X 0,Y 142.428,Z 596.022,A -85,B 0,C 180,E1 -27389.887,E2 -27389.887} C_VEL
LIN {X 0,Y 140.205,Z 608.393,A -85,B 0,C 180,E1 -27390.628,E2 -27390.628} C_VEL
LIN {X 0,Y 136.415,Z 621.882,A -85,B 0,C 180,E1 -27391.782,E2 -27391.782} C_VEL
LIN {X 0,Y 132.233,Z 632.991,A -85,B 0,C 180,E1 -27393.167,E2 -27393.167} C_VEL
LIN {X 0,Y 128.111,Z 641.986,A -85,B 0,C 180,E1 -27394.627,E2 -27394.627} C_VEL
LIN {X 0,Y 123.48,Z 650.708,A -85,B 0,C 180,E1 -27396.493,E2 -27396.493} C_VEL
LIN {X 0,Y 118.974,Z 658.123,A -85,B 0,C 180,E1 -27398.492,E2 -27398.492} C_VEL
LIN {X 0,Y 112.859,Z 666.914,A -85,B 0,C 180,E1 -27401.646,E2 -27401.646} C_VEL
LIN {X 0,Y 108.259,Z 672.901,A -85,B 0,C 180,E1 -27404.431,E2 -27404.431} C_VEL
LIN {X 0,Y 102.604,Z 679.656,A -85,B 0,C 180,E1 -27408.633,E2 -27408.633} C_VEL
LIN {X 0,Y 98.295,Z 684.489,A -85,B 0,C 180,E1 -27412.574,E2 -27412.574} C_VEL
LIN {X 0,Y 93.209,Z 689.582,A -85,B 0,C 180,E1 -27418.143,E2 -27418.143} C_VEL
LIN {X 0,Y 89.14,Z 693.549,A -85,B 0,C 180,E1 -27424.302,E2 -27424.302} C_VEL
LIN {X 0,Y 86.243,Z 696.493,A -85,B 0,C 180,E1 -27430.976,E2 -27430.976} C_VEL
LIN {X 0,Y 84.949,Z 698.001,A -85,B 0,C 180,E1 -27435.629,E2 -27435.629} C_VEL
LIN {X 0,Y 83.795,Z 699.542,A -85,B 0,C 180,E1 -27445.189,E2 -27445.189} C_VEL
LIN {X 0,Y 83.888,Z 699.83,A -85,B 0,C 180,E1 -27450,E2 -27450} C_VEL
LIN {X 0,Y 84.136,Z 698.938,A -85,B 0,C 180,E1 -27459.617,E2 -27459.617} C_VEL
LIN {X 0,Y 84.95,Z 698.001,A -85,B 0,C 180,E1 -27464.37,E2 -27464.37} C_VEL
LIN {X 0,Y 88.012,Z 694.64,A -85,B 0,C 180,E1 -27473.532,E2 -27473.532} C_VEL
LIN {X 0,Y 91.754,Z 691.011,A -85,B 0,C 180,E1 -27479.859,E2 -27479.859} C_VEL
LIN {X 0,Y 96.5,Z 686.279,A -85,B 0,C 180,E1 -27485.635,E2 -27485.635} C_VEL
LIN {X 0,Y 100.095,Z 682.491,A -85,B 0,C 180,E1 -27489.191,E2 -27489.191} C_VEL
LIN {X 0,Y 105.044,Z 676.836,A -85,B 0,C 180,E1 -27493.296,E2 -27493.296} C_VEL
LIN {X 0,Y 110.531,Z 670.034,A -85,B 0,C 180,E1 -27496.988,E2 -27496.988} C_VEL
LIN {X 0,Y 116.477,Z 661.821,A -85,B 0,C 180,E1 -27500.291,E2 -27500.291} C_VEL
LIN {X 0,Y 121.515,Z 654,A -85,B 0,C 180,E1 -27502.678,E2 -27502.678} C_VEL
LIN {X 0,Y 126.124,Z 645.923,A -85,B 0,C 180,E1 -27504.581,E2 -27504.581} C_VEL
LIN {X 0,Y 130.827,Z 636.167,A -85,B 0,C 180,E1 -27506.371,E2 -27506.371} C_VEL
LIN {X 0,Y 134.273,Z 627.782,A -85,B 0,C 180,E1 -27507.564,E2 -27507.564} C_VEL
LIN {X 0,Y 137.772,Z 617.28,A -85,B 0,C 180,E1 -27508.697,E2 -27508.697} C_VEL
LIN {X 0,Y 140.473,Z 606.952,A -85,B 0,C 180,E1 -27509.481,E2 -27509.481} C_VEL
LIN {X 0,Y 142.353,Z 596.698,A -85,B 0,C 180,E1 -27510.056,E2 -27510.056} C_VEL
LIN {X 0,Y 144.403,Z 577.013,A -85,B 0,C 180,E1 -27510.811,E2 -27510.811} C_VEL
LIN {X 0,Y 144.361,Z 575.543,A -85,B 0,C 180,E1 -27510.988,E2 -27510.988} C_VEL
LIN {X 0,Y 141.046,Z 565.171,A -85,B 0,C 180,E1 -27514.67,E2 -27514.67} C_VEL
LIN {X 0,Y 139.403,Z 561.062,A -85,B 0,C 180,E1 -27516.637,E2 -27516.637} C_VEL
LIN {X 0,Y 136.361,Z 555.416,A -85,B 0,C 180,E1 -27520.618,E2 -27520.618} C_VEL
LIN {X 0,Y 133.917,Z 551.33,A -85,B 0,C 180,E1 -27524.588,E2 -27524.588} C_VEL
LIN {X 0,Y 131.984,Z 547.805,A -85,B 0,C 180,E1 -27528.866,E2 -27528.866} C_VEL
LIN {X 0,Y 130.017,Z 543.376,A -85,B 0,C 180,E1 -27538.447,E2 -27538.447} C_VEL
LIN {X 0,Y 129.984,Z 543.161,A -85,B 0,C 180,E1 -27539.995,E2 -27539.995} C_VEL
LIN {X 0,Y 130.1,Z 543.949,A -85,B 0,C 180,E1 -27543.479,E2 -27543.479} C_VEL
LIN {X 0,Y 131.977,Z 547.819,A -85,B 0,C 180,E1 -27551.51,E2 -27551.51} C_VEL
LIN {X 0,Y 132.631,Z 548.898,A -85,B 0,C 180,E1 -27553.104,E2 -27553.104} C_VEL
LIN {X 0,Y 133.226,Z 550.73,A -85,B 0,C 180,E1 -27554.571,E2 -27554.571} C_VEL
LIN {X 0,Y 134.289,Z 555.739,A -85,B 0,C 180,E1 -27557.169,E2 -27557.169} C_VEL
LIN {X 0,Y 136.152,Z 564.291,A -85,B 0,C 180,E1 -27560.863,E2 -27560.863} C_VEL
LIN {X 0,Y 137.072,Z 566.715,A -85,B 0,C 180,E1 -27562.194,E2 -27562.194} C_VEL
LIN {X 0,Y 139.984,Z 573.071,A -85,B 0,C 180,E1 -27565.729,E2 -27565.729} C_VEL
LIN {X 0,Y 143.247,Z 581.079,A -85,B 0,C 180,E1 -27569.161,E2 -27569.161} C_VEL
LIN {X 0,Y 145.839,Z 589.044,A -85,B 0,C 180,E1 -27571.803,E2 -27571.803} C_VEL
LIN {X 0,Y 147.956,Z 598.686,A -85,B 0,C 180,E1 -27574.435,E2 -27574.435} C_VEL
LIN {X 0,Y 149.66,Z 607.767,A -85,B 0,C 180,E1 -27577.031,E2 -27577.031} C_VEL
LIN {X 0,Y 151.755,Z 618.104,A -85,B 0,C 180,E1 -27580.412,E2 -27580.412} C_VEL
LIN {X 0,Y 154.171,Z 627.768,A -85,B 0,C 180,E1 -27584.036,E2 -27584.036} C_VEL
LIN {X 0,Y 157.069,Z 636.756,A -85,B 0,C 180,E1 -27587.843,E2 -27587.843} C_VEL
LIN {X 0,Y 160.774,Z 645.223,A -85,B 0,C 180,E1 -27591.884,E2 -27591.884} C_VEL
LIN {X 0,Y 165.69,Z 653.429,A -85,B 0,C 180,E1 -27596.262,E2 -27596.262} C_VEL
LIN {X 0,Y 171.724,Z 660.723,A -85,B 0,C 180,E1 -27600.587,E2 -27600.587} C_VEL
LIN {X 0,Y 178.753,Z 667.08,A -85,B 0,C 180,E1 -27604.718,E2 -27604.718} C_VEL
LIN {X 0,Y 188.048,Z 673.172,A -85,B 0,C 180,E1 -27609.11,E2 -27609.11} C_VEL
LIN {X 0,Y 198.366,Z 678.082,A -85,B 0,C 180,E1 -27613.043,E2 -27613.043} C_VEL
LIN {X 0,Y 209.527,Z 682.025,A -85,B 0,C 180,E1 -27616.571,E2 -27616.571} C_VEL
LIN {X 0,Y 221.303,Z 685.27,A -85,B 0,C 180,E1 -27619.872,E2 -27619.872} C_VEL
LIN {X 0,Y 227.378,Z 686.696,A -85,B 0,C 180,E1 -27621.502,E2 -27621.502} C_VEL
LIN {X 0,Y 233.541,Z 687.997,A -85,B 0,C 180,E1 -27623.225,E2 -27623.225} C_VEL
LIN {X 0,Y 239.783,Z 689.27,A -85,B 0,C 180,E1 -27625.188,E2 -27625.188} C_VEL
LIN {X 0,Y 243.466,Z 689.97,A -85,B 0,C 180,E1 -27626.69,E2 -27626.69} C_VEL
LIN {X 0,Y 246.785,Z 690.483,A -85,B 0,C 180,E1 -27628.368,E2 -27628.368} C_VEL
LIN {X 0,Y 248.629,Z 690.64,A -85,B 0,C 180,E1 -27630,E2 -27630} C_VEL
LIN {X 0,Y 246.77,Z 690.483,A -85,B 0,C 180,E1 -27631.632,E2 -27631.632} C_VEL
LIN {X 0,Y 243.446,Z 689.97,A -85,B 0,C 180,E1 -27633.31,E2 -27633.31} C_VEL
LIN {X 0,Y 239.017,Z 689.127,A -85,B 0,C 180,E1 -27635.061,E2 -27635.061} C_VEL
LIN {X 0,Y 233.045,Z 687.888,A -85,B 0,C 180,E1 -27636.928,E2 -27636.928} C_VEL
LIN {X 0,Y 225.677,Z 686.303,A -85,B 0,C 180,E1 -27638.958,E2 -27638.958} C_VEL
LIN {X 0,Y 215.345,Z 683.738,A -85,B 0,C 180,E1 -27641.758,E2 -27641.758} C_VEL
LIN {X 0,Y 200.328,Z 678.839,A -85,B 0,C 180,E1 -27646.299,E2 -27646.299} C_VEL
LIN {X 0,Y 190.875,Z 674.663,A -85,B 0,C 180,E1 -27649.74,E2 -27649.74} C_VEL
LIN {X 0,Y 180.97,Z 668.719,A -85,B 0,C 180,E1 -27654.139,E2 -27654.139} C_VEL
LIN {X 0,Y 174.565,Z 663.484,A -85,B 0,C 180,E1 -27657.669,E2 -27657.669} C_VEL
LIN {X 0,Y 167.914,Z 656.342,A -85,B 0,C 180,E1 -27662.061,E2 -27662.061} C_VEL
LIN {X 0,Y 162.977,Z 649.219,A -85,B 0,C 180,E1 -27666.054,E2 -27666.054} C_VEL
LIN {X 0,Y 158.836,Z 641.155,A -85,B 0,C 180,E1 -27670.131,E2 -27670.131} C_VEL
LIN {X 0,Y 155.328,Z 631.655,A -85,B 0,C 180,E1 -27674.372,E2 -27674.372} C_VEL
LIN {X 0,Y 153.056,Z 623.495,A -85,B 0,C 180,E1 -27677.629,E2 -27677.629} C_VEL
LIN {X 0,Y 150.603,Z 612.67,A -85,B 0,C 180,E1 -27681.419,E2 -27681.419} C_VEL
LIN {X 0,Y 148.586,Z 602.22,A -85,B 0,C 180,E1 -27684.595,E2 -27684.595} C_VEL
LIN {X 0,Y 146.49,Z 591.335,A -85,B 0,C 180,E1 -27687.544,E2 -27687.544} C_VEL
LIN {X 0,Y 144.002,Z 583.221,A -85,B 0,C 180,E1 -27690.09,E2 -27690.09} C_VEL
LIN {X 0,Y 141.196,Z 575.926,A -85,B 0,C 180,E1 -27692.943,E2 -27692.943} C_VEL
LIN {X 0,Y 138.104,Z 568.951,A -85,B 0,C 180,E1 -27696.479,E2 -27696.479} C_VEL
LIN {X 0,Y 135.58,Z 563.779,A -85,B 0,C 180,E1 -27699.865,E2 -27699.865} C_VEL
LIN {X 0,Y 133.692,Z 560.262,A -85,B 0,C 180,E1 -27702.855,E2 -27702.855} C_VEL
LIN {X 0,Y 132.445,Z 557.922,A -85,B 0,C 180,E1 -27705.21,E2 -27705.21} C_VEL
LIN {X 0,Y 130.827,Z 554.678,A -85,B 0,C 180,E1 -27709.144,E2 -27709.144} C_VEL
LIN {X 0,Y 129.126,Z 550.435,A -85,B 0,C 180,E1 -27718.445,E2 -27718.445} C_VEL
LIN {X 0,Y 129.122,Z 550.326,A -85,B 0,C 180,E1 -27720.784,E2 -27720.784} C_VEL
LIN {X 0,Y 129.306,Z 551.765,A -85,B 0,C 180,E1 -27724.193,E2 -27724.193} C_VEL
LIN {X 0,Y 131.092,Z 555.212,A -85,B 0,C 180,E1 -27731.211,E2 -27731.211} C_VEL
LIN {X 0,Y 133.318,Z 559.466,A -85,B 0,C 180,E1 -27736.072,E2 -27736.072} C_VEL
LIN {X 0,Y 135.338,Z 563.293,A -85,B 0,C 180,E1 -27739.386,E2 -27739.386} C_VEL
LIN {X 0,Y 137.595,Z 567.784,A -85,B 0,C 180,E1 -27742.48,E2 -27742.48} C_VEL
LIN {X 0,Y 139.614,Z 574.22,A -85,B 0,C 180,E1 -27745.157,E2 -27745.157} C_VEL
LIN {X 0,Y 140.855,Z 578.584,A -85,B 0,C 180,E1 -27746.688,E2 -27746.688} C_VEL
LIN {X 0,Y 138.917,Z 596.6,A -85,B 0,C 180,E1 -27747.384,E2 -27747.384} C_VEL
LIN {X 0,Y 136.282,Z 610.105,A -85,B 0,C 180,E1 -27748.179,E2 -27748.179} C_VEL
LIN {X 0,Y 132.809,Z 621.686,A -85,B 0,C 180,E1 -27749.175,E2 -27749.175} C_VEL
LIN {X 0,Y 128.489,Z 632.795,A -85,B 0,C 180,E1 -27750.518,E2 -27750.518} C_VEL
LIN {X 0,Y 124.212,Z 641.789,A -85,B 0,C 180,E1 -27751.929,E2 -27751.929} C_VEL
LIN {X 0,Y 119.396,Z 650.512,A -85,B 0,C 180,E1 -27753.754,E2 -27753.754} C_VEL
LIN {X 0,Y 114.686,Z 657.927,A -85,B 0,C 180,E1 -27755.712,E2 -27755.712} C_VEL
LIN {X 0,Y 108.26,Z 666.717,A -85,B 0,C 180,E1 -27758.83,E2 -27758.83} C_VEL
LIN {X 0,Y 103.388,Z 672.703,A -85,B 0,C 180,E1 -27761.605,E2 -27761.605} C_VEL
LIN {X 0,Y 97.687,Z 679.125,A -85,B 0,C 180,E1 -27765.601,E2 -27765.601} C_VEL
LIN {X 0,Y 92.729,Z 684.292,A -85,B 0,C 180,E1 -27769.893,E2 -27769.893} C_VEL
LIN {X 0,Y 87.224,Z 689.384,A -85,B 0,C 180,E1 -27775.666,E2 -27775.666} C_VEL
LIN {X 0,Y 82.775,Z 693.352,A -85,B 0,C 180,E1 -27782.162,E2 -27782.162} C_VEL
LIN {X 0,Y 79.526,Z 696.296,A -85,B 0,C 180,E1 -27789.299,E2 -27789.299} C_VEL
LIN {X 0,Y 78.056,Z 697.804,A -85,B 0,C 180,E1 -27794.329,E2 -27794.329} C_VEL
LIN {X 0,Y 76.715,Z 699.346,A -85,B 0,C 180,E1 -27804.744,E2 -27804.744} C_VEL
LIN {X 0,Y 76.786,Z 699.634,A -85,B 0,C 180,E1 -27810,E2 -27810} C_VEL
LIN {X 0,Y 77.124,Z 698.741,A -85,B 0,C 180,E1 -27820.501,E2 -27820.501} C_VEL
LIN {X 0,Y 78.057,Z 697.804,A -85,B 0,C 180,E1 -27825.671,E2 -27825.671} C_VEL
LIN {X 0,Y 81.517,Z 694.443,A -85,B 0,C 180,E1 -27835.536,E2 -27835.536} C_VEL
LIN {X 0,Y 85.647,Z 690.814,A -85,B 0,C 180,E1 -27842.233,E2 -27842.233} C_VEL
LIN {X 0,Y 90.813,Z 686.082,A -85,B 0,C 180,E1 -27848.251,E2 -27848.251} C_VEL
LIN {X 0,Y 96.755,Z 680.111,A -85,B 0,C 180,E1 -27853.631,E2 -27853.631} C_VEL
LIN {X 0,Y 102.242,Z 674.016,A -85,B 0,C 180,E1 -27857.641,E2 -27857.641} C_VEL
LIN {X 0,Y 107.038,Z 668.277,A -85,B 0,C 180,E1 -27860.487,E2 -27860.487} C_VEL
LIN {X 0,Y 112.065,Z 661.625,A -85,B 0,C 180,E1 -27863.091,E2 -27863.091} C_VEL
LIN {X 0,Y 117.335,Z 653.803,A -85,B 0,C 180,E1 -27865.444,E2 -27865.444} C_VEL
LIN {X 0,Y 122.138,Z 645.726,A -85,B 0,C 180,E1 -27867.302,E2 -27867.302} C_VEL
LIN {X 0,Y 127.034,Z 635.971,A -85,B 0,C 180,E1 -27869.038,E2 -27869.038} C_VEL
LIN {X 0,Y 130.607,Z 627.586,A -85,B 0,C 180,E1 -27870.19,E2 -27870.19} C_VEL
LIN {X 0,Y 134.224,Z 617.084,A -85,B 0,C 180,E1 -27871.286,E2 -27871.286} C_VEL
LIN {X 0,Y 137.107,Z 606.355,A -85,B 0,C 180,E1 -27872.051,E2 -27872.051} C_VEL
LIN {X 0,Y 139.039,Z 595.749,A -85,B 0,C 180,E1 -27872.631,E2 -27872.631} C_VEL
LIN {X 0,Y 140.852,Z 578.608,A -85,B 0,C 180,E1 -27873.312,E2 -27873.312} C_VEL
LIN {X 0,Y 138.335,Z 569.963,A -85,B 0,C 180,E1 -27876.519,E2 -27876.519} C_VEL
LIN {X 0,Y 137.034,Z 566.597,A -85,B 0,C 180,E1 -27878.25,E2 -27878.25} C_VEL
LIN {X 0,Y 134.388,Z 561.396,A -85,B 0,C 180,E1 -27882.102,E2 -27882.102} C_VEL
LIN {X 0,Y 132.546,Z 558.035,A -85,B 0,C 180,E1 -27885.408,E2 -27885.408} C_VEL
LIN {X 0,Y 130.787,Z 554.625,A -85,B 0,C 180,E1 -27889.644,E2 -27889.644} C_VEL
LIN {X 0,Y 129.149,Z 550.448,A -85,B 0,C 180,E1 -27898.436,E2 -27898.436} C_VEL
LIN {X 0,Y 129.117,Z 550.218,A -85,B 0,C 180,E1 -27899.995,E2 -27899.995} C_VEL
LIN {X 0,Y 129.191,Z 550.976,A -85,B 0,C 180,E1 -27903.114,E2 -27903.114} C_VEL
LIN {X 0,Y 131.092,Z 555.234,A -85,B 0,C 180,E1 -27911.605,E2 -27911.605} C_VEL
LIN {X 0,Y 133.314,Z 559.47,A -85,B 0,C 180,E1 -27916.456,E2 -27916.456} C_VEL
LIN {X 0,Y 135.509,Z 563.645,A -85,B 0,C 180,E1 -27920.032,E2 -27920.032} C_VEL
LIN {X 0,Y 137.072,Z 566.715,A -85,B 0,C 180,E1 -27922.194,E2 -27922.194} C_VEL
LIN {X 0,Y 138.393,Z 570.515,A -85,B 0,C 180,E1 -27923.987,E2 -27923.987} C_VEL
LIN {X 0,Y 139.39,Z 575.173,A -85,B 0,C 180,E1 -27925.454,E2 -27925.454} C_VEL
LIN {X 0,Y 140.965,Z 585.557,A -85,B 0,C 180,E1 -27927.922,E2 -27927.922} C_VEL
LIN {X 0,Y 142.105,Z 592.278,A -85,B 0,C 180,E1 -27929.701,E2 -27929.701} C_VEL
LIN {X 0,Y 143.579,Z 600.217,A -85,B 0,C 180,E1 -27932.053,E2 -27932.053} C_VEL
LIN {X 0,Y 144.992,Z 610.369,A -85,B 0,C 180,E1 -27935.094,E2 -27935.094} C_VEL
LIN {X 0,Y 146.322,Z 618.959,A -85,B 0,C 180,E1 -27938.024,E2 -27938.024} C_VEL
LIN {X 0,Y 148.085,Z 628.286,A -85,B 0,C 180,E1 -27941.632,E2 -27941.632} C_VEL
LIN {X 0,Y 150.259,Z 637.015,A -85,B 0,C 180,E1 -27945.446,E2 -27945.446} C_VEL
LIN {X 0,Y 153.122,Z 645.243,A -85,B 0,C 180,E1 -27949.501,E2 -27949.501} C_VEL
LIN {X 0,Y 156.924,Z 652.844,A -85,B 0,C 180,E1 -27953.714,E2 -27953.714} C_VEL
LIN {X 0,Y 161.322,Z 659.274,A -85,B 0,C 180,E1 -27957.627,E2 -27957.627} C_VEL
LIN {X 0,Y 168.235,Z 666.692,A -85,B 0,C 180,E1 -27962.644,E2 -27962.644} C_VEL
LIN {X 0,Y 175.723,Z 672.379,A -85,B 0,C 180,E1 -27966.898,E2 -27966.898} C_VEL
LIN {X 0,Y 185.456,Z 677.681,A -85,B 0,C 180,E1 -27971.321,E2 -27971.321} C_VEL
LIN {X 0,Y 197.154,Z 682.157,A -85,B 0,C 180,E1 -27975.55,E2 -27975.55} C_VEL
LIN {X 0,Y 207.784,Z 685.144,A -85,B 0,C 180,E1 -27978.76,E2 -27978.76} C_VEL
LIN {X 0,Y 219.948,Z 687.776,A -85,B 0,C 180,E1 -27982.087,E2 -27982.087} C_VEL
LIN {X 0,Y 226.207,Z 688.864,A -85,B 0,C 180,E1 -27983.797,E2 -27983.797} C_VEL
LIN {X 0,Y 232.563,Z 689.853,A -85,B 0,C 180,E1 -27985.705,E2 -27985.705} C_VEL
LIN {X 0,Y 234.935,Z 690.204,A -85,B 0,C 180,E1 -27986.57,E2 -27986.57} C_VEL
LIN {X 0,Y 239.034,Z 690.703,A -85,B 0,C 180,E1 -27988.372,E2 -27988.372} C_VEL
LIN {X 0,Y 241.27,Z 690.843,A -85,B 0,C 180,E1 -27990,E2 -27990} C_VEL
LIN {X 0,Y 238.865,Z 690.698,A -85,B 0,C 180,E1 -27991.686,E2 -27991.686} C_VEL
LIN {X 0,Y 234.899,Z 690.205,A -85,B 0,C 180,E1 -27993.431,E2 -27993.431} C_VEL
LIN {X 0,Y 232.562,Z 689.855,A -85,B 0,C 180,E1 -27994.291,E2 -27994.291} C_VEL
LIN {X 0,Y 226.208,Z 688.862,A -85,B 0,C 180,E1 -27996.206,E2 -27996.206} C_VEL
LIN {X 0,Y 219.956,Z 687.763,A -85,B 0,C 180,E1 -27997.927,E2 -27997.927} C_VEL
LIN {X 0,Y 205.752,Z 684.645,A -85,B 0,C 180,E1 -28001.826,E2 -28001.826} C_VEL
LIN {X 0,Y 190.724,Z 679.874,A -85,B 0,C 180,E1 -28006.663,E2 -28006.663} C_VEL
LIN {X 0,Y 180.456,Z 675.141,A -85,B 0,C 180,E1 -28010.832,E2 -28010.832} C_VEL
LIN {X 0,Y 173.065,Z 670.607,A -85,B 0,C 180,E1 -28014.489,E2 -28014.489} C_VEL
LIN {X 0,Y 165.265,Z 663.835,A -85,B 0,C 180,E1 -28019.343,E2 -28019.343} C_VEL
LIN {X 0,Y 159.164,Z 656.462,A -85,B 0,C 180,E1 -28024.123,E2 -28024.123} C_VEL
LIN {X 0,Y 154.836,Z 648.99,A -85,B 0,C 180,E1 -28028.474,E2 -28028.474} C_VEL
LIN {X 0,Y 151.85,Z 641.872,A -85,B 0,C 180,E1 -28032.231,E2 -28032.231} C_VEL
LIN {X 0,Y 148.932,Z 631.986,A -85,B 0,C 180,E1 -28036.807,E2 -28036.807} C_VEL
LIN {X 0,Y 146.991,Z 622.816,A -85,B 0,C 180,E1 -28040.549,E2 -28040.549} C_VEL
LIN {X 0,Y 145.361,Z 612.799,A -85,B 0,C 180,E1 -28044.114,E2 -28044.114} C_VEL
LIN {X 0,Y 143.902,Z 602.412,A -85,B 0,C 180,E1 -28047.318,E2 -28047.318} C_VEL
LIN {X 0,Y 142.299,Z 592.941,A -85,B 0,C 180,E1 -28050.103,E2 -28050.103} C_VEL
LIN {X 0,Y 139.886,Z 584.738,A -85,B 0,C 180,E1 -28053.022,E2 -28053.022} C_VEL
LIN {X 0,Y 136.82,Z 576.887,A -85,B 0,C 180,E1 -28056.697,E2 -28056.697} C_VEL
LIN {X 0,Y 134.209,Z 570.873,A -85,B 0,C 180,E1 -28060.395,E2 -28060.395} C_VEL
LIN {X 0,Y 132.101,Z 566.667,A -85,B 0,C 180,E1 -28063.984,E2 -28063.984} C_VEL
LIN {X 0,Y 130.94,Z 564.327,A -85,B 0,C 180,E1 -28066.423,E2 -28066.423} C_VEL
LIN {X 0,Y 129.667,Z 561.51,A -85,B 0,C 180,E1 -28069.891,E2 -28069.891} C_VEL
LIN {X 0,Y 128.258,Z 557.508,A -85,B 0,C 180,E1 -28078.435,E2 -28078.435} C_VEL
LIN {X 0,Y 128.257,Z 557.371,A -85,B 0,C 180,E1 -28080.79,E2 -28080.79} C_VEL
LIN {X 0,Y 129.894,Z 562.018,A -85,B 0,C 180,E1 -28090.428,E2 -28090.428} C_VEL
LIN {X 0,Y 131.735,Z 565.817,A -85,B 0,C 180,E1 -28094.882,E2 -28094.882} C_VEL
LIN {X 0,Y 133.83,Z 570.133,A -85,B 0,C 180,E1 -28098.631,E2 -28098.631} C_VEL
LIN {X 0,Y 135.526,Z 574.002,A -85,B 0,C 180,E1 -28101.189,E2 -28101.189} C_VEL
LIN {X 0,Y 137.409,Z 580.846,A -85,B 0,C 180,E1 -28103.983,E2 -28103.983} C_VEL
LIN {X 0,Y 137.544,Z 581.408,A -85,B 0,C 180,E1 -28104.177,E2 -28104.177} C_VEL
LIN {X 0,Y 135.555,Z 598.044,A -85,B 0,C 180,E1 -28104.791,E2 -28104.791} C_VEL
LIN {X 0,Y 132.516,Z 611.843,A -85,B 0,C 180,E1 -28105.633,E2 -28105.633} C_VEL
LIN {X 0,Y 129.493,Z 621.489,A -85,B 0,C 180,E1 -28106.427,E2 -28106.427} C_VEL
LIN {X 0,Y 125.037,Z 632.599,A -85,B 0,C 180,E1 -28107.717,E2 -28107.717} C_VEL
LIN {X 0,Y 120.609,Z 641.593,A -85,B 0,C 180,E1 -28109.067,E2 -28109.067} C_VEL
LIN {X 0,Y 115.593,Z 650.315,A -85,B 0,C 180,E1 -28110.82,E2 -28110.82} C_VEL
LIN {X 0,Y 110.69,Z 657.731,A -85,B 0,C 180,E1 -28112.725,E2 -28112.725} C_VEL
LIN {X 0,Y 103.944,Z 666.52,A -85,B 0,C 180,E1 -28115.772,E2 -28115.772} C_VEL
LIN {X 0,Y 98.807,Z 672.507,A -85,B 0,C 180,E1 -28118.519,E2 -28118.519} C_VEL
LIN {X 0,Y 92.828,Z 678.819,A -85,B 0,C 180,E1 -28122.426,E2 -28122.426} C_VEL
LIN {X 0,Y 87.393,Z 684.095,A -85,B 0,C 180,E1 -28126.879,E2 -28126.879} C_VEL
LIN {X 0,Y 81.43,Z 689.187,A -85,B 0,C 180,E1 -28132.833,E2 -28132.833} C_VEL
LIN {X 0,Y 76.549,Z 693.156,A -85,B 0,C 180,E1 -28139.672,E2 -28139.672} C_VEL
LIN {X 0,Y 72.898,Z 696.099,A -85,B 0,C 180,E1 -28147.317,E2 -28147.317} C_VEL
LIN {X 0,Y 71.22,Z 697.607,A -85,B 0,C 180,E1 -28152.78,E2 -28152.78} C_VEL
LIN {X 0,Y 69.628,Z 699.149,A -85,B 0,C 180,E1 -28164.207,E2 -28164.207} C_VEL
LIN {X 0,Y 69.683,Z 699.438,A -85,B 0,C 180,E1 -28170,E2 -28170} C_VEL
LIN {X 0,Y 70.146,Z 698.545,A -85,B 0,C 180,E1 -28181.559,E2 -28181.559} C_VEL
LIN {X 0,Y 71.221,Z 697.607,A -85,B 0,C 180,E1 -28187.219,E2 -28187.219} C_VEL
LIN {X 0,Y 75.143,Z 694.245,A -85,B 0,C 180,E1 -28197.881,E2 -28197.881} C_VEL
LIN {X 0,Y 79.71,Z 690.617,A -85,B 0,C 180,E1 -28204.967,E2 -28204.967} C_VEL
LIN {X 0,Y 85.339,Z 685.885,A -85,B 0,C 180,E1 -28211.21,E2 -28211.21} C_VEL
LIN {X 0,Y 91.7,Z 679.913,A -85,B 0,C 180,E1 -28216.723,E2 -28216.723} C_VEL
LIN {X 0,Y 97.581,Z 673.819,A -85,B 0,C 180,E1 -28220.735,E2 -28220.735} C_VEL
LIN {X 0,Y 102.645,Z 668.08,A -85,B 0,C 180,E1 -28223.562,E2 -28223.562} C_VEL
LIN {X 0,Y 107.947,Z 661.428,A -85,B 0,C 180,E1 -28226.108,E2 -28226.108} C_VEL
LIN {X 0,Y 113.457,Z 653.607,A -85,B 0,C 180,E1 -28228.399,E2 -28228.399} C_VEL
LIN {X 0,Y 118.444,Z 645.53,A -85,B 0,C 180,E1 -28230.202,E2 -28230.202} C_VEL
LIN {X 0,Y 123.53,Z 635.775,A -85,B 0,C 180,E1 -28231.864,E2 -28231.864} C_VEL
LIN {X 0,Y 127.23,Z 627.39,A -85,B 0,C 180,E1 -28232.963,E2 -28232.963} C_VEL
LIN {X 0,Y 130.96,Z 616.888,A -85,B 0,C 180,E1 -28234.012,E2 -28234.012} C_VEL
LIN {X 0,Y 133.93,Z 606.131,A -85,B 0,C 180,E1 -28234.738,E2 -28234.738} C_VEL
LIN {X 0,Y 135.81,Z 596.305,A -85,B 0,C 180,E1 -28235.266,E2 -28235.266} C_VEL
LIN {X 0,Y 137.517,Z 581.282,A -85,B 0,C 180,E1 -28235.863,E2 -28235.863} C_VEL
LIN {X 0,Y 135.527,Z 573.999,A -85,B 0,C 180,E1 -28238.811,E2 -28238.811} C_VEL
LIN {X 0,Y 133.733,Z 569.911,A -85,B 0,C 180,E1 -28241.529,E2 -28241.529} C_VEL
LIN {X 0,Y 131.825,Z 566.033,A -85,B 0,C 180,E1 -28244.931,E2 -28244.931} C_VEL
LIN {X 0,Y 130.395,Z 563.234,A -85,B 0,C 180,E1 -28248.137,E2 -28248.137} C_VEL
LIN {X 0,Y 129.549,Z 561.365,A -85,B 0,C 180,E1 -28250.629,E2 -28250.629} C_VEL
LIN {X 0,Y 128.256,Z 557.382,A -85,B 0,C 180,E1 -28259.21,E2 -28259.21} C_VEL
LIN {X 0,Y 128.269,Z 557.613,A -85,B 0,C 180,E1 -28261.958,E2 -28261.958} C_VEL
LIN {X 0,Y 129.877,Z 562.013,A -85,B 0,C 180,E1 -28270.776,E2 -28270.776} C_VEL
LIN {X 0,Y 131.821,Z 566.051,A -85,B 0,C 180,E1 -28275.455,E2 -28275.455} C_VEL
LIN {X 0,Y 133.622,Z 569.716,A -85,B 0,C 180,E1 -28278.686,E2 -28278.686} C_VEL
LIN {X 0,Y 135.81,Z 574.533,A -85,B 0,C 180,E1 -28281.956,E2 -28281.956} C_VEL
LIN {X 0,Y 138.544,Z 581.178,A -85,B 0,C 180,E1 -28285.437,E2 -28285.437} C_VEL
LIN {X 0,Y 141.095,Z 588.565,A -85,B 0,C 180,E1 -28288.439,E2 -28288.439} C_VEL
LIN {X 0,Y 142.105,Z 592.278,A -85,B 0,C 180,E1 -28289.701,E2 -28289.701} C_VEL
LIN {X 0,Y 142.501,Z 595.751,A -85,B 0,C 180,E1 -28290.462,E2 -28290.462} C_VEL
LIN {X 0,Y 141.682,Z 602.209,A -85,B 0,C 180,E1 -28291.19,E2 -28291.19} C_VEL
LIN {X 0,Y 140.657,Z 608.658,A -85,B 0,C 180,E1 -28291.957,E2 -28291.957} C_VEL
LIN {X 0,Y 140.429,Z 612.125,A -85,B 0,C 180,E1 -28292.76,E2 -28292.76} C_VEL
LIN {X 0,Y 141.325,Z 621.071,A -85,B 0,C 180,E1 -28295.947,E2 -28295.947} C_VEL
LIN {X 0,Y 142.325,Z 628.702,A -85,B 0,C 180,E1 -28299.013,E2 -28299.013} C_VEL
LIN {X 0,Y 143.949,Z 637.753,A -85,B 0,C 180,E1 -28303.113,E2 -28303.113} C_VEL
LIN {X 0,Y 146.076,Z 645.597,A -85,B 0,C 180,E1 -28307.138,E2 -28307.138} C_VEL
LIN {X 0,Y 148.647,Z 652.277,A -85,B 0,C 180,E1 -28310.923,E2 -28310.923} C_VEL
LIN {X 0,Y 152.979,Z 659.839,A -85,B 0,C 180,E1 -28315.777,E2 -28315.777} C_VEL
LIN {X 0,Y 158.89,Z 666.978,A -85,B 0,C 180,E1 -28320.886,E2 -28320.886} C_VEL
LIN {X 0,Y 165.925,Z 672.886,A -85,B 0,C 180,E1 -28325.583,E2 -28325.583} C_VEL
LIN {X 0,Y 175.284,Z 678.292,A -85,B 0,C 180,E1 -28330.417,E2 -28330.417} C_VEL
LIN {X 0,Y 185.682,Z 682.478,A -85,B 0,C 180,E1 -28334.636,E2 -28334.636} C_VEL
LIN {X 0,Y 194.311,Z 685.07,A -85,B 0,C 180,E1 -28337.551,E2 -28337.551} C_VEL
LIN {X 0,Y 206.312,Z 687.69,A -85,B 0,C 180,E1 -28341.048,E2 -28341.048} C_VEL
LIN {X 0,Y 219.066,Z 689.685,A -85,B 0,C 180,E1 -28344.477,E2 -28344.477} C_VEL
LIN {X 0,Y 225.812,Z 690.454,A -85,B 0,C 180,E1 -28346.431,E2 -28346.431} C_VEL
LIN {X 0,Y 230.637,Z 690.921,A -85,B 0,C 180,E1 -28348.254,E2 -28348.254} C_VEL
LIN {X 0,Y 231.958,Z 690.982,A -85,B 0,C 180,E1 -28348.833,E2 -28348.833} C_VEL
LIN {X 0,Y 233.784,Z 691.05,A -85,B 0,C 180,E1 -28350,E2 -28350} C_VEL
LIN {X 0,Y 231.957,Z 690.984,A -85,B 0,C 180,E1 -28351.15,E2 -28351.15} C_VEL
LIN {X 0,Y 230.603,Z 690.922,A -85,B 0,C 180,E1 -28351.746,E2 -28351.746} C_VEL
LIN {X 0,Y 225.353,Z 690.406,A -85,B 0,C 180,E1 -28353.705,E2 -28353.705} C_VEL
LIN {X 0,Y 218.89,Z 689.659,A -85,B 0,C 180,E1 -28355.575,E2 -28355.575} C_VEL
LIN {X 0,Y 206.308,Z 687.696,A -85,B 0,C 180,E1 -28358.945,E2 -28358.945} C_VEL
LIN {X 0,Y 194.017,Z 684.977,A -85,B 0,C 180,E1 -28362.553,E2 -28362.553} C_VEL
LIN {X 0,Y 180.408,Z 680.558,A -85,B 0,C 180,E1 -28367.383,E2 -28367.383} C_VEL
LIN {X 0,Y 170.843,Z 675.982,A -85,B 0,C 180,E1 -28371.73,E2 -28371.73} C_VEL
LIN {X 0,Y 163.833,Z 671.304,A -85,B 0,C 180,E1 -28375.741,E2 -28375.741} C_VEL
LIN {X 0,Y 156.188,Z 664.073,A -85,B 0,C 180,E1 -28381.255,E2 -28381.255} C_VEL
LIN {X 0,Y 151.486,Z 657.573,A -85,B 0,C 180,E1 -28385.727,E2 -28385.727} C_VEL
LIN {X 0,Y 147.656,Z 650.006,A -85,B 0,C 180,E1 -28390.406,E2 -28390.406} C_VEL
LIN {X 0,Y 144.754,Z 641.037,A -85,B 0,C 180,E1 -28395.258,E2 -28395.258} C_VEL
LIN {X 0,Y 142.896,Z 632.347,A -85,B 0,C 180,E1 -28399.412,E2 -28399.412} C_VEL
LIN {X 0,Y 141.515,Z 622.739,A -85,B 0,C 180,E1 -28403.426,E2 -28403.426} C_VEL
LIN {X 0,Y 140.634,Z 613.828,A -85,B 0,C 180,E1 -28406.659,E2 -28406.659} C_VEL
LIN {X 0,Y 139.613,Z 603.02,A -85,B 0,C 180,E1 -28410.093,E2 -28410.093} C_VEL
LIN {X 0,Y 138.427,Z 595.001,A -85,B 0,C 180,E1 -28412.714,E2 -28412.714} C_VEL
LIN {X 0,Y 136.407,Z 587.681,A -85,B 0,C 180,E1 -28415.664,E2 -28415.664} C_VEL
LIN {X 0,Y 133.765,Z 580.492,A -85,B 0,C 180,E1 -28419.435,E2 -28419.435} C_VEL
LIN {X 0,Y 131.841,Z 575.878,A -85,B 0,C 180,E1 -28422.637,E2 -28422.637} C_VEL
LIN {X 0,Y 129.889,Z 571.433,A -85,B 0,C 180,E1 -28426.711,E2 -28426.711} C_VEL
LIN {X 0,Y 128.435,Z 568.231,A -85,B 0,C 180,E1 -28430.954,E2 -28430.954} C_VEL
LIN {X 0,Y 127.377,Z 564.443,A -85,B 0,C 180,E1 -28439.215,E2 -28439.215} C_VEL
LIN {X 0,Y 127.385,Z 564.511,A -85,B 0,C 180,E1 -28440.894,E2 -28440.894} C_VEL
LIN {X 0,Y 128.719,Z 568.831,A -85,B 0,C 180,E1 -28449.63,E2 -28449.63} C_VEL
LIN {X 0,Y 130.343,Z 572.474,A -85,B 0,C 180,E1 -28453.963,E2 -28453.963} C_VEL
LIN {X 0,Y 132.364,Z 576.969,A -85,B 0,C 180,E1 -28457.881,E2 -28457.881} C_VEL
LIN {X 0,Y 133.505,Z 580.104,A -85,B 0,C 180,E1 -28459.814,E2 -28459.814} C_VEL
LIN {X 0,Y 134.449,Z 584.122,A -85,B 0,C 180,E1 -28461.468,E2 -28461.468} C_VEL
LIN {X 0,Y 132.879,Z 596.931,A -85,B 0,C 180,E1 -28461.974,E2 -28461.974} C_VEL
LIN {X 0,Y 129.598,Z 611.646,A -85,B 0,C 180,E1 -28462.797,E2 -28462.797} C_VEL
LIN {X 0,Y 126.45,Z 621.4,A -85,B 0,C 180,E1 -28463.555,E2 -28463.555} C_VEL
LIN {X 0,Y 121.897,Z 632.402,A -85,B 0,C 180,E1 -28464.761,E2 -28464.761} C_VEL
LIN {X 0,Y 117.325,Z 641.397,A -85,B 0,C 180,E1 -28466.036,E2 -28466.036} C_VEL
LIN {X 0,Y 112.118,Z 650.118,A -85,B 0,C 180,E1 -28467.7,E2 -28467.7} C_VEL
LIN {X 0,Y 107.017,Z 657.534,A -85,B 0,C 180,E1 -28469.525,E2 -28469.525} C_VEL
LIN {X 0,Y 99.946,Z 666.323,A -85,B 0,C 180,E1 -28472.455,E2 -28472.455} C_VEL
LIN {X 0,Y 94.542,Z 672.31,A -85,B 0,C 180,E1 -28475.145,E2 -28475.145} C_VEL
LIN {X 0,Y 88.17,Z 678.62,A -85,B 0,C 180,E1 -28478.999,E2 -28478.999} C_VEL
LIN {X 0,Y 81.555,Z 684.521,A -85,B 0,C 180,E1 -28484.152,E2 -28484.152} C_VEL
LIN {X 0,Y 75.872,Z 688.99,A -85,B 0,C 180,E1 -28489.579,E2 -28489.579} C_VEL
LIN {X 0,Y 70.496,Z 692.959,A -85,B 0,C 180,E1 -28496.749,E2 -28496.749} C_VEL
LIN {X 0,Y 66.359,Z 695.901,A -85,B 0,C 180,E1 -28504.936,E2 -28504.936} C_VEL
LIN {X 0,Y 64.456,Z 697.411,A -85,B 0,C 180,E1 -28510.907,E2 -28510.907} C_VEL
LIN {X 0,Y 62.561,Z 698.953,A -85,B 0,C 180,E1 -28523.55,E2 -28523.55} C_VEL
LIN {X 0,Y 62.574,Z 699.241,A -85,B 0,C 180,E1 -28530,E2 -28530} C_VEL
LIN {X 0,Y 63.182,Z 698.348,A -85,B 0,C 180,E1 -28542.854,E2 -28542.854} C_VEL
LIN {X 0,Y 64.457,Z 697.411,A -85,B 0,C 180,E1 -28549.093,E2 -28549.093} C_VEL
LIN {X 0,Y 68.926,Z 694.048,A -85,B 0,C 180,E1 -28560.652,E2 -28560.652} C_VEL
LIN {X 0,Y 73.985,Z 690.42,A -85,B 0,C 180,E1 -28568.13,E2 -28568.13} C_VEL
LIN {X 0,Y 80.107,Z 685.688,A -85,B 0,C 180,E1 -28574.576,E2 -28574.576} C_VEL
LIN {X 0,Y 85.786,Z 680.807,A -85,B 0,C 180,E1 -28579.27,E2 -28579.27} C_VEL
LIN {X 0,Y 91.938,Z 674.933,A -85,B 0,C 180,E1 -28583.383,E2 -28583.383} C_VEL
LIN {X 0,Y 97.24,Z 669.444,A -85,B 0,C 180,E1 -28586.217,E2 -28586.217} C_VEL
LIN {X 0,Y 104.15,Z 661.232,A -85,B 0,C 180,E1 -28589.357,E2 -28589.357} C_VEL
LIN {X 0,Y 109.905,Z 653.411,A -85,B 0,C 180,E1 -28591.551,E2 -28591.551} C_VEL
LIN {X 0,Y 115.083,Z 645.334,A -85,B 0,C 180,E1 -28593.269,E2 -28593.269} C_VEL
LIN {X 0,Y 120.345,Z 635.579,A -85,B 0,C 180,E1 -28594.846,E2 -28594.846} C_VEL
LIN {X 0,Y 124.154,Z 627.221,A -85,B 0,C 180,E1 -28595.879,E2 -28595.879} C_VEL
LIN {X 0,Y 127.948,Z 616.899,A -85,B 0,C 180,E1 -28596.85,E2 -28596.85} C_VEL
LIN {X 0,Y 130.995,Z 606.243,A -85,B 0,C 180,E1 -28597.523,E2 -28597.523} C_VEL
LIN {X 0,Y 133.101,Z 595.477,A -85,B 0,C 180,E1 -28598.055,E2 -28598.055} C_VEL
LIN {X 0,Y 134.449,Z 584.124,A -85,B 0,C 180,E1 -28598.532,E2 -28598.532} C_VEL
LIN {X 0,Y 133.121,Z 578.802,A -85,B 0,C 180,E1 -28600.851,E2 -28600.851} C_VEL
LIN {X 0,Y 131.003,Z 573.951,A -85,B 0,C 180,E1 -28604.635,E2 -28604.635} C_VEL
LIN {X 0,Y 129.647,Z 571.024,A -85,B 0,C 180,E1 -28607.671,E2 -28607.671} C_VEL
LIN {X 0,Y 128.437,Z 568.215,A -85,B 0,C 180,E1 -28611.341,E2 -28611.341} C_VEL
LIN {X 0,Y 127.385,Z 564.416,A -85,B 0,C 180,E1 -28619.402,E2 -28619.402} C_VEL
LIN {X 0,Y 127.383,Z 564.64,A -85,B 0,C 180,E1 -28621.576,E2 -28621.576} C_VEL
LIN {X 0,Y 128.726,Z 568.872,A -85,B 0,C 180,E1 -28630.05,E2 -28630.05} C_VEL
LIN {X 0,Y 130.35,Z 572.566,A -85,B 0,C 180,E1 -28634.385,E2 -28634.385} C_VEL
LIN {X 0,Y 132.035,Z 576.272,A -85,B 0,C 180,E1 -28637.703,E2 -28637.703} C_VEL
LIN {X 0,Y 134.371,Z 582.02,A -85,B 0,C 180,E1 -28641.471,E2 -28641.471} C_VEL
LIN {X 0,Y 136.812,Z 589.08,A -85,B 0,C 180,E1 -28644.968,E2 -28644.968} C_VEL
LIN {X 0,Y 138.753,Z 596.539,A -85,B 0,C 180,E1 -28647.83,E2 -28647.83} C_VEL
LIN {X 0,Y 139.996,Z 606.267,A -85,B 0,C 180,E1 -28650.88,E2 -28650.88} C_VEL
LIN {X 0,Y 140.429,Z 612.125,A -85,B 0,C 180,E1 -28652.76,E2 -28652.76} C_VEL
LIN {X 0,Y 140.529,Z 616.97,A -85,B 0,C 180,E1 -28654.153,E2 -28654.153} C_VEL
LIN {X 0,Y 139.345,Z 625.463,A -85,B 0,C 180,E1 -28656.201,E2 -28656.201} C_VEL
LIN {X 0,Y 137.962,Z 633.525,A -85,B 0,C 180,E1 -28658.473,E2 -28658.473} C_VEL
LIN {X 0,Y 137.838,Z 637.69,A -85,B 0,C 180,E1 -28660.186,E2 -28660.186} C_VEL
LIN {X 0,Y 139.45,Z 646.504,A -85,B 0,C 180,E1 -28664.869,E2 -28664.869} C_VEL
LIN {X 0,Y 141.716,Z 653.824,A -85,B 0,C 180,E1 -28669.287,E2 -28669.287} C_VEL
LIN {X 0,Y 144.636,Z 659.882,A -85,B 0,C 180,E1 -28673.361,E2 -28673.361} C_VEL
LIN {X 0,Y 149.899,Z 667.259,A -85,B 0,C 180,E1 -28678.954,E2 -28678.954} C_VEL
LIN {X 0,Y 156.314,Z 673.279,A -85,B 0,C 180,E1 -28684.045,E2 -28684.045} C_VEL
LIN {X 0,Y 165.193,Z 678.859,A -85,B 0,C 180,E1 -28689.373,E2 -28689.373} C_VEL
LIN {X 0,Y 175.425,Z 683.14,A -85,B 0,C 180,E1 -28694.035,E2 -28694.035} C_VEL
LIN {X 0,Y 186.716,Z 686.375,A -85,B 0,C 180,E1 -28698.117,E2 -28698.117} C_VEL
LIN {X 0,Y 199.462,Z 688.815,A -85,B 0,C 180,E1 -28701.898,E2 -28701.898} C_VEL
LIN {X 0,Y 211.584,Z 690.365,A -85,B 0,C 180,E1 -28705.15,E2 -28705.15} C_VEL
LIN {X 0,Y 218.158,Z 690.96,A -85,B 0,C 180,E1 -28706.975,E2 -28706.975} C_VEL
LIN {X 0,Y 221.888,Z 691.158,A -85,B 0,C 180,E1 -28708.185,E2 -28708.185} C_VEL
LIN {X 0,Y 224.898,Z 691.239,A -85,B 0,C 180,E1 -28709.317,E2 -28709.317} C_VEL
LIN {X 0,Y 226.136,Z 691.262,A -85,B 0,C 180,E1 -28710,E2 -28710} C_VEL
LIN {X 0,Y 224.897,Z 691.24,A -85,B 0,C 180,E1 -28710.669,E2 -28710.669} C_VEL
LIN {X 0,Y 221.877,Z 691.158,A -85,B 0,C 180,E1 -28711.815,E2 -28711.815} C_VEL
LIN {X 0,Y 218.159,Z 690.959,A -85,B 0,C 180,E1 -28713.027,E2 -28713.027} C_VEL
LIN {X 0,Y 207.973,Z 689.995,A -85,B 0,C 180,E1 -28715.819,E2 -28715.819} C_VEL
LIN {X 0,Y 192.696,Z 687.667,A -85,B 0,C 180,E1 -28720.045,E2 -28720.045} C_VEL
LIN {X 0,Y 180.952,Z 684.919,A -85,B 0,C 180,E1 -28723.855,E2 -28723.855} C_VEL
LIN {X 0,Y 170.177,Z 681.163,A -85,B 0,C 180,E1 -28728.235,E2 -28728.235} C_VEL
LIN {X 0,Y 160.588,Z 676.237,A -85,B 0,C 180,E1 -28733.224,E2 -28733.224} C_VEL
LIN {X 0,Y 153.81,Z 671.191,A -85,B 0,C 180,E1 -28737.801,E2 -28737.801} C_VEL
LIN {X 0,Y 147.367,Z 664.214,A -85,B 0,C 180,E1 -28743.437,E2 -28743.437} C_VEL
LIN {X 0,Y 143.31,Z 657.441,A -85,B 0,C 180,E1 -28748.32,E2 -28748.32} C_VEL
LIN {X 0,Y 140.265,Z 649.441,A -85,B 0,C 180,E1 -28753.414,E2 -28753.414} C_VEL
LIN {X 0,Y 138.505,Z 641.929,A -85,B 0,C 180,E1 -28757.66,E2 -28757.66} C_VEL
LIN {X 0,Y 137.296,Z 632.888,A -85,B 0,C 180,E1 -28762.108,E2 -28762.108} C_VEL
LIN {X 0,Y 136.587,Z 623.721,A -85,B 0,C 180,E1 -28766.055,E2 -28766.055} C_VEL
LIN {X 0,Y 136.129,Z 613.651,A -85,B 0,C 180,E1 -28769.783,E2 -28769.783} C_VEL
LIN {X 0,Y 135.575,Z 603.129,A -85,B 0,C 180,E1 -28773.24,E2 -28773.24} C_VEL
LIN {X 0,Y 134.602,Z 596.367,A -85,B 0,C 180,E1 -28775.829,E2 -28775.829} C_VEL
LIN {X 0,Y 132.752,Z 589.36,A -85,B 0,C 180,E1 -28779.169,E2 -28779.169} C_VEL
LIN {X 0,Y 130.644,Z 583.242,A -85,B 0,C 180,E1 -28782.997,E2 -28782.997} C_VEL
LIN {X 0,Y 128.608,Z 578.154,A -85,B 0,C 180,E1 -28787.57,E2 -28787.57} C_VEL
LIN {X 0,Y 127.295,Z 574.974,A -85,B 0,C 180,E1 -28791.872,E2 -28791.872} C_VEL
LIN {X 0,Y 126.51,Z 571.476,A -85,B 0,C 180,E1 -28799.378,E2 -28799.378} C_VEL
LIN {X 0,Y 126.508,Z 571.547,A -85,B 0,C 180,E1 -28800.539,E2 -28800.539} C_VEL
LIN {X 0,Y 127.549,Z 575.531,A -85,B 0,C 180,E1 -28808.72,E2 -28808.72} C_VEL
LIN {X 0,Y 129.018,Z 579.254,A -85,B 0,C 180,E1 -28813.117,E2 -28813.117} C_VEL
LIN {X 0,Y 130.69,Z 583.364,A -85,B 0,C 180,E1 -28816.705,E2 -28816.705} C_VEL
LIN {X 0,Y 131.463,Z 585.865,A -85,B 0,C 180,E1 -28818.209,E2 -28818.209} C_VEL
LIN {X 0,Y 131.719,Z 587.076,A -85,B 0,C 180,E1 -28818.741,E2 -28818.741} C_VEL
LIN {X 0,Y 129.495,Z 601.457,A -85,B 0,C 180,E1 -28819.305,E2 -28819.305} C_VEL
LIN {X 0,Y 126.563,Z 612.874,A -85,B 0,C 180,E1 -28819.936,E2 -28819.936} C_VEL
LIN {X 0,Y 123.602,Z 621.652,A -85,B 0,C 180,E1 -28820.582,E2 -28820.582} C_VEL
LIN {X 0,Y 119.102,Z 632.206,A -85,B 0,C 180,E1 -28821.663,E2 -28821.663} C_VEL
LIN {X 0,Y 114.386,Z 641.201,A -85,B 0,C 180,E1 -28822.838,E2 -28822.838} C_VEL
LIN {X 0,Y 108.998,Z 649.922,A -85,B 0,C 180,E1 -28824.392,E2 -28824.392} C_VEL
LIN {X 0,Y 103.691,Z 657.337,A -85,B 0,C 180,E1 -28826.097,E2 -28826.097} C_VEL
LIN {X 0,Y 96.311,Z 666.126,A -85,B 0,C 180,E1 -28828.878,E2 -28828.878} C_VEL
LIN {X 0,Y 90.624,Z 672.113,A -85,B 0,C 180,E1 -28831.455,E2 -28831.455} C_VEL
LIN {X 0,Y 83.853,Z 678.423,A -85,B 0,C 180,E1 -28835.198,E2 -28835.198} C_VEL
LIN {X 0,Y 77.633,Z 683.639,A -85,B 0,C 180,E1 -28839.557,E2 -28839.557} C_VEL
LIN {X 0,Y 70.602,Z 688.793,A -85,B 0,C 180,E1 -28845.829,E2 -28845.829} C_VEL
LIN {X 0,Y 64.665,Z 692.762,A -85,B 0,C 180,E1 -28853.291,E2 -28853.291} C_VEL
LIN {X 0,Y 59.962,Z 695.704,A -85,B 0,C 180,E1 -28862.042,E2 -28862.042} C_VEL
LIN {X 0,Y 57.766,Z 697.214,A -85,B 0,C 180,E1 -28868.593,E2 -28868.593} C_VEL
LIN {X 0,Y 55.496,Z 698.756,A -85,B 0,C 180,E1 -28882.725,E2 -28882.725} C_VEL
LIN {X 0,Y 55.486,Z 699.045,A -85,B 0,C 180,E1 -28890,E2 -28890} C_VEL
LIN {X 0,Y 56.271,Z 698.151,A -85,B 0,C 180,E1 -28904.465,E2 -28904.465} C_VEL
LIN {X 0,Y 57.767,Z 697.214,A -85,B 0,C 180,E1 -28911.406,E2 -28911.406} C_VEL
LIN {X 0,Y 62.907,Z 693.852,A -85,B 0,C 180,E1 -28923.959,E2 -28923.959} C_VEL
LIN {X 0,Y 68.512,Z 690.223,A -85,B 0,C 180,E1 -28931.818,E2 -28931.818} C_VEL
LIN {X 0,Y 75.19,Z 685.491,A -85,B 0,C 180,E1 -28938.396,E2 -28938.396} C_VEL
LIN {X 0,Y 81.29,Z 680.609,A -85,B 0,C 180,E1 -28943.102,E2 -28943.102} C_VEL
LIN {X 0,Y 87.873,Z 674.736,A -85,B 0,C 180,E1 -28947.116,E2 -28947.116} C_VEL
LIN {X 0,Y 93.457,Z 669.247,A -85,B 0,C 180,E1 -28949.859,E2 -28949.859} C_VEL
LIN {X 0,Y 100.713,Z 661.035,A -85,B 0,C 180,E1 -28952.838,E2 -28952.838} C_VEL
LIN {X 0,Y 106.711,Z 653.215,A -85,B 0,C 180,E1 -28954.9,E2 -28954.9} C_VEL
LIN {X 0,Y 112.071,Z 645.138,A -85,B 0,C 180,E1 -28956.51,E2 -28956.51} C_VEL
LIN {X 0,Y 117.504,Z 635.383,A -85,B 0,C 180,E1 -28957.98,E2 -28957.98} C_VEL
LIN {X 0,Y 121.381,Z 627.136,A -85,B 0,C 180,E1 -28958.927,E2 -28958.927} C_VEL
LIN {X 0,Y 125.056,Z 617.565,A -85,B 0,C 180,E1 -28959.775,E2 -28959.775} C_VEL
LIN {X 0,Y 128.452,Z 605.98,A -85,B 0,C 180,E1 -28960.468,E2 -28960.468} C_VEL
LIN {X 0,Y 130.655,Z 595.012,A -85,B 0,C 180,E1 -28960.952,E2 -28960.952} C_VEL
LIN {X 0,Y 131.717,Z 587.093,A -85,B 0,C 180,E1 -28961.258,E2 -28961.258} C_VEL
LIN {X 0,Y 130.934,Z 584.048,A -85,B 0,C 180,E1 -28962.825,E2 -28962.825} C_VEL
LIN {X 0,Y 129.373,Z 580.104,A -85,B 0,C 180,E1 -28966.043,E2 -28966.043} C_VEL
LIN {X 0,Y 128.067,Z 576.993,A -85,B 0,C 180,E1 -28969.468,E2 -28969.468} C_VEL
LIN {X 0,Y 127.346,Z 575.06,A -85,B 0,C 180,E1 -28972.065,E2 -28972.065} C_VEL
LIN {X 0,Y 126.52,Z 571.369,A -85,B 0,C 180,E1 -28979.995,E2 -28979.995} C_VEL
LIN {X 0,Y 126.508,Z 572.361,A -85,B 0,C 180,E1 -28982.582,E2 -28982.582} C_VEL
LIN {X 0,Y 127.547,Z 575.55,A -85,B 0,C 180,E1 -28989.11,E2 -28989.11} C_VEL
LIN {X 0,Y 129.085,Z 579.442,A -85,B 0,C 180,E1 -28993.675,E2 -28993.675} C_VEL
LIN {X 0,Y 130.695,Z 583.342,A -85,B 0,C 180,E1 -28997.097,E2 -28997.097} C_VEL
LIN {X 0,Y 132.705,Z 589.38,A -85,B 0,C 180,E1 -29000.839,E2 -29000.839} C_VEL
LIN {X 0,Y 134.559,Z 596.126,A -85,B 0,C 180,E1 -29004.077,E2 -29004.077} C_VEL
LIN {X 0,Y 135.583,Z 603.094,A -85,B 0,C 180,E1 -29006.759,E2 -29006.759} C_VEL
LIN {X 0,Y 136.125,Z 613.663,A -85,B 0,C 180,E1 -29010.217,E2 -29010.217} C_VEL
LIN {X 0,Y 136.749,Z 625.582,A -85,B 0,C 180,E1 -29014.686,E2 -29014.686} C_VEL
LIN {X 0,Y 137.715,Z 636.587,A -85,B 0,C 180,E1 -29019.632,E2 -29019.632} C_VEL
LIN {X 0,Y 137.838,Z 637.69,A -85,B 0,C 180,E1 -29020.186,E2 -29020.186} C_VEL
LIN {X 0,Y 137.919,Z 640.474,A -85,B 0,C 180,E1 -29021.417,E2 -29021.417} C_VEL
LIN {X 0,Y 137.134,Z 646.28,A -85,B 0,C 180,E1 -29023.706,E2 -29023.706} C_VEL
LIN {X 0,Y 135.657,Z 655.573,A -85,B 0,C 180,E1 -29027.882,E2 -29027.882} C_VEL
LIN {X 0,Y 136.237,Z 658.807,A -85,B 0,C 180,E1 -29029.897,E2 -29029.897} C_VEL
LIN {X 0,Y 141.195,Z 667.541,A -85,B 0,C 180,E1 -29036.803,E2 -29036.803} C_VEL
LIN {X 0,Y 146.882,Z 673.594,A -85,B 0,C 180,E1 -29042.261,E2 -29042.261} C_VEL
LIN {X 0,Y 154.784,Z 679.104,A -85,B 0,C 180,E1 -29047.87,E2 -29047.87} C_VEL
LIN {X 0,Y 163.378,Z 683.106,A -85,B 0,C 180,E1 -29052.475,E2 -29052.475} C_VEL
LIN {X 0,Y 173.334,Z 686.28,A -85,B 0,C 180,E1 -29056.662,E2 -29056.662} C_VEL
LIN {X 0,Y 187.616,Z 689.141,A -85,B 0,C 180,E1 -29061.383,E2 -29061.383} C_VEL
LIN {X 0,Y 197.781,Z 690.467,A -85,B 0,C 180,E1 -29064.206,E2 -29064.206} C_VEL
LIN {X 0,Y 204.837,Z 691.03,A -85,B 0,C 180,E1 -29066.065,E2 -29066.065} C_VEL
LIN {X 0,Y 212.415,Z 691.415,A -85,B 0,C 180,E1 -29068.104,E2 -29068.104} C_VEL
LIN {X 0,Y 218.049,Z 691.485,A -85,B 0,C 180,E1 -29070,E2 -29070} C_VEL
LIN {X 0,Y 210.996,Z 691.382,A -85,B 0,C 180,E1 -29072.298,E2 -29072.298} C_VEL
LIN {X 0,Y 204.318,Z 690.984,A -85,B 0,C 180,E1 -29074.086,E2 -29074.086} C_VEL
LIN {X 0,Y 191.395,Z 689.678,A -85,B 0,C 180,E1 -29077.533,E2 -29077.533} C_VEL
LIN {X 0,Y 179.03,Z 687.586,A -85,B 0,C 180,E1 -29081.319,E2 -29081.319} C_VEL
LIN {X 0,Y 167.777,Z 684.643,A -85,B 0,C 180,E1 -29085.557,E2 -29085.557} C_VEL
LIN {X 0,Y 157.569,Z 680.553,A -85,B 0,C 180,E1 -29090.516,E2 -29090.516} C_VEL
LIN {X 0,Y 150.776,Z 676.571,A -85,B 0,C 180,E1 -29094.803,E2 -29094.803} C_VEL
LIN {X 0,Y 145.08,Z 671.957,A -85,B 0,C 180,E1 -29099.323,E2 -29099.323} C_VEL
LIN {X 0,Y 139.574,Z 665.264,A -85,B 0,C 180,E1 -29105.117,E2 -29105.117} C_VEL
LIN {X 0,Y 136.077,Z 658.408,A -85,B 0,C 180,E1 -29110.386,E2 -29110.386} C_VEL
LIN {X 0,Y 133.627,Z 649.768,A -85,B 0,C 180,E1 -29116.135,E2 -29116.135} C_VEL
LIN {X 0,Y 132.434,Z 641.231,A -85,B 0,C 180,E1 -29121.078,E2 -29121.078} C_VEL
LIN {X 0,Y 132.015,Z 632.864,A -85,B 0,C 180,E1 -29125.275,E2 -29125.275} C_VEL
LIN {X 0,Y 131.983,Z 624.289,A -85,B 0,C 180,E1 -29129.022,E2 -29129.022} C_VEL
LIN {X 0,Y 132.122,Z 614.151,A -85,B 0,C 180,E1 -29132.825,E2 -29132.825} C_VEL
LIN {X 0,Y 131.982,Z 605.042,A -85,B 0,C 180,E1 -29136.05,E2 -29136.05} C_VEL
LIN {X 0,Y 131.067,Z 598.103,A -85,B 0,C 180,E1 -29139.094,E2 -29139.094} C_VEL
LIN {X 0,Y 129.6,Z 591.859,A -85,B 0,C 180,E1 -29142.652,E2 -29142.652} C_VEL
LIN {X 0,Y 128.192,Z 587.26,A -85,B 0,C 180,E1 -29146.127,E2 -29146.127} C_VEL
LIN {X 0,Y 126.795,Z 583.513,A -85,B 0,C 180,E1 -29150.232,E2 -29150.232} C_VEL
LIN {X 0,Y 126.186,Z 581.749,A -85,B 0,C 180,E1 -29152.806,E2 -29152.806} C_VEL
LIN {X 0,Y 125.645,Z 578.502,A -85,B 0,C 180,E1 -29160.005,E2 -29160.005} C_VEL
LIN {X 0,Y 126.451,Z 582.423,A -85,B 0,C 180,E1 -29167.992,E2 -29167.992} C_VEL
LIN {X 0,Y 127.673,Z 585.894,A -85,B 0,C 180,E1 -29172.119,E2 -29172.119} C_VEL
LIN {X 0,Y 129.008,Z 589.595,A -85,B 0,C 180,E1 -29175.406,E2 -29175.406} C_VEL
LIN {X 0,Y 129.196,Z 590.238,A -85,B 0,C 180,E1 -29175.853,E2 -29175.853} C_VEL
LIN {X 0,Y 127.206,Z 601.76,A -85,B 0,C 180,E1 -29176.309,E2 -29176.309} C_VEL
LIN {X 0,Y 124.316,Z 612.711,A -85,B 0,C 180,E1 -29176.868,E2 -29176.868} C_VEL
LIN {X 0,Y 121.076,Z 621.971,A -85,B 0,C 180,E1 -29177.483,E2 -29177.483} C_VEL
LIN {X 0,Y 116.668,Z 632.01,A -85,B 0,C 180,E1 -29178.421,E2 -29178.421} C_VEL
LIN {X 0,Y 111.824,Z 641.005,A -85,B 0,C 180,E1 -29179.486,E2 -29179.486} C_VEL
LIN {X 0,Y 106.261,Z 649.726,A -85,B 0,C 180,E1 -29180.901,E2 -29180.901} C_VEL
LIN {X 0,Y 100.764,Z 657.141,A -85,B 0,C 180,E1 -29182.461,E2 -29182.461} C_VEL
LIN {X 0,Y 93.085,Z 665.93,A -85,B 0,C 180,E1 -29185.042,E2 -29185.042} C_VEL
LIN {X 0,Y 87.124,Z 671.917,A -85,B 0,C 180,E1 -29187.461,E2 -29187.461} C_VEL
LIN {X 0,Y 79.953,Z 678.226,A -85,B 0,C 180,E1 -29191.015,E2 -29191.015} C_VEL
LIN {X 0,Y 72.575,Z 683.932,A -85,B 0,C 180,E1 -29195.759,E2 -29195.759} C_VEL
LIN {X 0,Y 65.686,Z 688.597,A -85,B 0,C 180,E1 -29201.501,E2 -29201.501} C_VEL
LIN {X 0,Y 59.095,Z 692.565,A -85,B 0,C 180,E1 -29209.149,E2 -29209.149} C_VEL
LIN {X 0,Y 53.757,Z 695.506,A -85,B 0,C 180,E1 -29218.47,E2 -29218.47} C_VEL
LIN {X 0,Y 51.179,Z 697.016,A -85,B 0,C 180,E1 -29225.672,E2 -29225.672} C_VEL
LIN {X 0,Y 48.443,Z 698.559,A -85,B 0,C 180,E1 -29241.658,E2 -29241.658} C_VEL
LIN {X 0,Y 48.381,Z 698.849,A -85,B 0,C 180,E1 -29250,E2 -29250} C_VEL
LIN {X 0,Y 49.396,Z 697.954,A -85,B 0,C 180,E1 -29266.532,E2 -29266.532} C_VEL
LIN {X 0,Y 51.179,Z 697.016,A -85,B 0,C 180,E1 -29274.328,E2 -29274.328} C_VEL
LIN {X 0,Y 57.145,Z 693.655,A -85,B 0,C 180,E1 -29287.946,E2 -29287.946} C_VEL
LIN {X 0,Y 63.364,Z 690.025,A -85,B 0,C 180,E1 -29296.132,E2 -29296.132} C_VEL
LIN {X 0,Y 70.655,Z 685.294,A -85,B 0,C 180,E1 -29302.726,E2 -29302.726} C_VEL
LIN {X 0,Y 77.209,Z 680.411,A -85,B 0,C 180,E1 -29307.35,E2 -29307.35} C_VEL
LIN {X 0,Y 84.221,Z 674.539,A -85,B 0,C 180,E1 -29311.185,E2 -29311.185} C_VEL
LIN {X 0,Y 90.086,Z 669.049,A -85,B 0,C 180,E1 -29313.787,E2 -29313.787} C_VEL
LIN {X 0,Y 97.662,Z 660.838,A -85,B 0,C 180,E1 -29316.564,E2 -29316.564} C_VEL
LIN {X 0,Y 103.895,Z 653.018,A -85,B 0,C 180,E1 -29318.452,E2 -29318.452} C_VEL
LIN {X 0,Y 109.439,Z 644.942,A -85,B 0,C 180,E1 -29319.915,E2 -29319.915} C_VEL
LIN {X 0,Y 115.034,Z 635.187,A -85,B 0,C 180,E1 -29321.256,E2 -29321.256} C_VEL
LIN {X 0,Y 119.651,Z 625.37,A -85,B 0,C 180,E1 -29322.264,E2 -29322.264} C_VEL
LIN {X 0,Y 123.372,Z 615.523,A -85,B 0,C 180,E1 -29323.01,E2 -29323.01} C_VEL
LIN {X 0,Y 126.42,Z 605.121,A -85,B 0,C 180,E1 -29323.525,E2 -29323.525} C_VEL
LIN {X 0,Y 128.41,Z 595.498,A -85,B 0,C 180,E1 -29323.922,E2 -29323.922} C_VEL
LIN {X 0,Y 129.176,Z 590.261,A -85,B 0,C 180,E1 -29324.137,E2 -29324.137} C_VEL
LIN {X 0,Y 127.817,Z 586.285,A -85,B 0,C 180,E1 -29327.491,E2 -29327.491} C_VEL
LIN {X 0,Y 126.592,Z 582.861,A -85,B 0,C 180,E1 -29331.415,E2 -29331.415} C_VEL
LIN {X 0,Y 126.106,Z 581.544,A -85,B 0,C 180,E1 -29333.596,E2 -29333.596} C_VEL
LIN {X 0,Y 125.646,Z 578.491,A -85,B 0,C 180,E1 -29339.995,E2 -29339.995} C_VEL
LIN {X 0,Y 126.449,Z 582.446,A -85,B 0,C 180,E1 -29348.384,E2 -29348.384} C_VEL
LIN {X 0,Y 127.747,Z 586.084,A -85,B 0,C 180,E1 -29352.707,E2 -29352.707} C_VEL
LIN {X 0,Y 129.032,Z 590.025,A -85,B 0,C 180,E1 -29356.102,E2 -29356.102} C_VEL
LIN {X 0,Y 130.631,Z 595.911,A -85,B 0,C 180,E1 -29359.746,E2 -29359.746} C_VEL
LIN {X 0,Y 131.649,Z 602.077,A -85,B 0,C 180,E1 -29362.765,E2 -29362.765} C_VEL
LIN {X 0,Y 132.155,Z 608.697,A -85,B 0,C 180,E1 -29365.305,E2 -29365.305} C_VEL
LIN {X 0,Y 132.032,Z 619.236,A -85,B 0,C 180,E1 -29369.012,E2 -29369.012} C_VEL
LIN {X 0,Y 131.96,Z 628.629,A -85,B 0,C 180,E1 -29372.814,E2 -29372.814} C_VEL
LIN {X 0,Y 132.212,Z 637.769,A -85,B 0,C 180,E1 -29377.123,E2 -29377.123} C_VEL
LIN {X 0,Y 133.024,Z 646.414,A -85,B 0,C 180,E1 -29381.831,E2 -29381.831} C_VEL
LIN {X 0,Y 134.728,Z 654.482,A -85,B 0,C 180,E1 -29386.904,E2 -29386.904} C_VEL
LIN {X 0,Y 136.237,Z 658.807,A -85,B 0,C 180,E1 -29389.897,E2 -29389.897} C_VEL
LIN {X 0,Y 136.956,Z 661.945,A -85,B 0,C 180,E1 -29391.985,E2 -29391.985} C_VEL
LIN {X 0,Y 136.831,Z 667.472,A -85,B 0,C 180,E1 -29395.449,E2 -29395.449} C_VEL
LIN {X 0,Y 137.197,Z 672.49,A -85,B 0,C 180,E1 -29399.01,E2 -29399.01} C_VEL
LIN {X 0,Y 138.673,Z 674.739,A -85,B 0,C 180,E1 -29401.16,E2 -29401.16} C_VEL
LIN {X 0,Y 145.41,Z 679.733,A -85,B 0,C 180,E1 -29406.668,E2 -29406.668} C_VEL
LIN {X 0,Y 152.694,Z 683.41,A -85,B 0,C 180,E1 -29411.205,E2 -29411.205} C_VEL
LIN {X 0,Y 160.138,Z 686.094,A -85,B 0,C 180,E1 -29414.892,E2 -29414.892} C_VEL
LIN {X 0,Y 171.589,Z 688.811,A -85,B 0,C 180,E1 -29419.397,E2 -29419.397} C_VEL
LIN {X 0,Y 184.533,Z 690.651,A -85,B 0,C 180,E1 -29423.439,E2 -29423.439} C_VEL
LIN {X 0,Y 197.082,Z 691.581,A -85,B 0,C 180,E1 -29426.779,E2 -29426.779} C_VEL
LIN {X 0,Y 203.865,Z 691.723,A -85,B 0,C 180,E1 -29428.538,E2 -29428.538} C_VEL
LIN {X 0,Y 208.901,Z 691.738,A -85,B 0,C 180,E1 -29430,E2 -29430} C_VEL
LIN {X 0,Y 201.83,Z 691.701,A -85,B 0,C 180,E1 -29431.996,E2 -29431.996} C_VEL
LIN {X 0,Y 190.45,Z 691.13,A -85,B 0,C 180,E1 -29434.939,E2 -29434.939} C_VEL
LIN {X 0,Y 175.79,Z 689.466,A -85,B 0,C 180,E1 -29439.202,E2 -29439.202} C_VEL
LIN {X 0,Y 165.729,Z 687.505,A -85,B 0,C 180,E1 -29442.768,E2 -29442.768} C_VEL
LIN {X 0,Y 154.854,Z 684.247,A -85,B 0,C 180,E1 -29447.637,E2 -29447.637} C_VEL
LIN {X 0,Y 146.549,Z 680.377,A -85,B 0,C 180,E1 -29452.56,E2 -29452.56} C_VEL
LIN {X 0,Y 141.148,Z 676.86,A -85,B 0,C 180,E1 -29456.623,E2 -29456.623} C_VEL
LIN {X 0,Y 135.69,Z 671.778,A -85,B 0,C 180,E1 -29461.906,E2 -29461.906} C_VEL
LIN {X 0,Y 131.368,Z 665.182,A -85,B 0,C 180,E1 -29467.908,E2 -29467.908} C_VEL
LIN {X 0,Y 128.888,Z 658.577,A -85,B 0,C 180,E1 -29473.221,E2 -29473.221} C_VEL
LIN {X 0,Y 127.477,Z 650.92,A -85,B 0,C 180,E1 -29478.587,E2 -29478.587} C_VEL
LIN {X 0,Y 127.032,Z 642.785,A -85,B 0,C 180,E1 -29483.513,E2 -29483.513} C_VEL
LIN {X 0,Y 127.221,Z 633.203,A -85,B 0,C 180,E1 -29488.477,E2 -29488.477} C_VEL
LIN {X 0,Y 127.876,Z 623.203,A -85,B 0,C 180,E1 -29492.825,E2 -29492.825} C_VEL
LIN {X 0,Y 128.526,Z 613.963,A -85,B 0,C 180,E1 -29496.3,E2 -29496.3} C_VEL
LIN {X 0,Y 128.669,Z 608.938,A -85,B 0,C 180,E1 -29498.209,E2 -29498.209} C_VEL
LIN {X 0,Y 128.166,Z 602.568,A -85,B 0,C 180,E1 -29501.212,E2 -29501.212} C_VEL
LIN {X 0,Y 127.27,Z 596.606,A -85,B 0,C 180,E1 -29504.901,E2 -29504.901} C_VEL
LIN {X 0,Y 126.176,Z 592.425,A -85,B 0,C 180,E1 -29508.56,E2 -29508.56} C_VEL
LIN {X 0,Y 125.189,Z 588.748,A -85,B 0,C 180,E1 -29513.154,E2 -29513.154} C_VEL
LIN {X 0,Y 124.76,Z 585.708,A -85,B 0,C 180,E1 -29520.005,E2 -29520.005} C_VEL
LIN {X 0,Y 125.385,Z 589.41,A -85,B 0,C 180,E1 -29527.452,E2 -29527.452} C_VEL
LIN {X 0,Y 126.291,Z 592.606,A -85,B 0,C 180,E1 -29531.236,E2 -29531.236} C_VEL
LIN {X 0,Y 126.772,Z 594.365,A -85,B 0,C 180,E1 -29532.89,E2 -29532.89} C_VEL
LIN {X 0,Y 124.29,Z 606.17,A -85,B 0,C 180,E1 -29533.388,E2 -29533.388} C_VEL
LIN {X 0,Y 120.206,Z 619.229,A -85,B 0,C 180,E1 -29534.067,E2 -29534.067} C_VEL
LIN {X 0,Y 115.456,Z 630.226,A -85,B 0,C 180,E1 -29534.91,E2 -29534.91} C_VEL
LIN {X 0,Y 109.663,Z 640.809,A -85,B 0,C 180,E1 -29535.992,E2 -29535.992} C_VEL
LIN {X 0,Y 103.936,Z 649.529,A -85,B 0,C 180,E1 -29537.235,E2 -29537.235} C_VEL
LIN {X 0,Y 98.267,Z 656.944,A -85,B 0,C 180,E1 -29538.626,E2 -29538.626} C_VEL
LIN {X 0,Y 90.305,Z 665.733,A -85,B 0,C 180,E1 -29540.951,E2 -29540.951} C_VEL
LIN {X 0,Y 84.082,Z 671.72,A -85,B 0,C 180,E1 -29543.158,E2 -29543.158} C_VEL
LIN {X 0,Y 76.525,Z 678.029,A -85,B 0,C 180,E1 -29546.438,E2 -29546.438} C_VEL
LIN {X 0,Y 67.877,Z 684.228,A -85,B 0,C 180,E1 -29551.419,E2 -29551.419} C_VEL
LIN {X 0,Y 61.206,Z 688.4,A -85,B 0,C 180,E1 -29556.508,E2 -29556.508} C_VEL
LIN {X 0,Y 53.904,Z 692.368,A -85,B 0,C 180,E1 -29564.186,E2 -29564.186} C_VEL
LIN {X 0,Y 47.817,Z 695.309,A -85,B 0,C 180,E1 -29573.991,E2 -29573.991} C_VEL
LIN {X 0,Y 44.772,Z 696.819,A -85,B 0,C 180,E1 -29581.906,E2 -29581.906} C_VEL
LIN {X 0,Y 41.424,Z 698.363,A -85,B 0,C 180,E1 -29600.232,E2 -29600.232} C_VEL
LIN {X 0,Y 41.293,Z 698.653,A -85,B 0,C 180,E1 -29610,E2 -29610} C_VEL
LIN {X 0,Y 42.614,Z 697.757,A -85,B 0,C 180,E1 -29629.259,E2 -29629.259} C_VEL
LIN {X 0,Y 44.773,Z 696.819,A -85,B 0,C 180,E1 -29638.093,E2 -29638.093} C_VEL
LIN {X 0,Y 51.721,Z 693.459,A -85,B 0,C 180,E1 -29652.797,E2 -29652.797} C_VEL
LIN {X 0,Y 58.641,Z 689.828,A -85,B 0,C 180,E1 -29661.169,E2 -29661.169} C_VEL
LIN {X 0,Y 63.875,Z 686.887,A -85,B 0,C 180,E1 -29665.608,E2 -29665.608} C_VEL
LIN {X 0,Y 72.178,Z 681.308,A -85,B 0,C 180,E1 -29671.202,E2 -29671.202} C_VEL
LIN {X 0,Y 79.513,Z 675.653,A -85,B 0,C 180,E1 -29674.954,E2 -29674.954} C_VEL
LIN {X 0,Y 87.176,Z 668.853,A -85,B 0,C 180,E1 -29677.987,E2 -29677.987} C_VEL
LIN {X 0,Y 95.055,Z 660.641,A -85,B 0,C 180,E1 -29680.505,E2 -29680.505} C_VEL
LIN {X 0,Y 101.503,Z 652.822,A -85,B 0,C 180,E1 -29682.18,E2 -29682.18} C_VEL
LIN {X 0,Y 107.211,Z 644.746,A -85,B 0,C 180,E1 -29683.476,E2 -29683.476} C_VEL
LIN {X 0,Y 112.955,Z 634.991,A -85,B 0,C 180,E1 -29684.664,E2 -29684.664} C_VEL
LIN {X 0,Y 117.559,Z 625.47,A -85,B 0,C 180,E1 -29685.534,E2 -29685.534} C_VEL
LIN {X 0,Y 121.486,Z 615.327,A -85,B 0,C 180,E1 -29686.217,E2 -29686.217} C_VEL
LIN {X 0,Y 124.637,Z 604.77,A -85,B 0,C 180,E1 -29686.65,E2 -29686.65} C_VEL
LIN {X 0,Y 126.752,Z 594.396,A -85,B 0,C 180,E1 -29687.07,E2 -29687.07} C_VEL
LIN {X 0,Y 125.643,Z 590.488,A -85,B 0,C 180,E1 -29691.147,E2 -29691.147} C_VEL
LIN {X 0,Y 125.138,Z 588.54,A -85,B 0,C 180,E1 -29693.95,E2 -29693.95} C_VEL
LIN {X 0,Y 124.758,Z 585.722,A -85,B 0,C 180,E1 -29700.399,E2 -29700.399} C_VEL
LIN {X 0,Y 125.264,Z 589.14,A -85,B 0,C 180,E1 -29707.45,E2 -29707.45} C_VEL
LIN {X 0,Y 126.185,Z 592.602,A -85,B 0,C 180,E1 -29711.643,E2 -29711.643} C_VEL
LIN {X 0,Y 127.319,Z 596.933,A -85,B 0,C 180,E1 -29715.298,E2 -29715.298} C_VEL
LIN {X 0,Y 128.231,Z 603.166,A -85,B 0,C 180,E1 -29719.089,E2 -29719.089} C_VEL
LIN {X 0,Y 128.671,Z 608.938,A -85,B 0,C 180,E1 -29721.794,E2 -29721.794} C_VEL
LIN {X 0,Y 128.349,Z 617.505,A -85,B 0,C 180,E1 -29724.963,E2 -29724.963} C_VEL
LIN {X 0,Y 127.538,Z 628.252,A -85,B 0,C 180,E1 -29729.273,E2 -29729.273} C_VEL
LIN {X 0,Y 127.026,Z 638.015,A -85,B 0,C 180,E1 -29733.912,E2 -29733.912} C_VEL
LIN {X 0,Y 127.085,Z 646.2,A -85,B 0,C 180,E1 -29738.466,E2 -29738.466} C_VEL
LIN {X 0,Y 127.915,Z 654.339,A -85,B 0,C 180,E1 -29743.72,E2 -29743.72} C_VEL
LIN {X 0,Y 130.015,Z 662.106,A -85,B 0,C 180,E1 -29749.56,E2 -29749.56} C_VEL
LIN {X 0,Y 133.286,Z 668.433,A -85,B 0,C 180,E1 -29755.005,E2 -29755.005} C_VEL
LIN {X 0,Y 137.69,Z 673.823,A -85,B 0,C 180,E1 -29760.184,E2 -29760.184} C_VEL
LIN {X 0,Y 138.673,Z 674.739,A -85,B 0,C 180,E1 -29761.16,E2 -29761.16} C_VEL
LIN {X 0,Y 140.369,Z 677.039,A -85,B 0,C 180,E1 -29763.313,E2 -29763.313} C_VEL
LIN {X 0,Y 143.699,Z 683.565,A -85,B 0,C 180,E1 -29769.869,E2 -29769.869} C_VEL
LIN {X 0,Y 145.929,Z 685.148,A -85,B 0,C 180,E1 -29771.917,E2 -29771.917} C_VEL
LIN {X 0,Y 146.941,Z 685.595,A -85,B 0,C 180,E1 -29772.546,E2 -29772.546} C_VEL
LIN {X 0,Y 158.139,Z 688.732,A -85,B 0,C 180,E1 -29777.861,E2 -29777.861} C_VEL
LIN {X 0,Y 172.598,Z 690.985,A -85,B 0,C 180,E1 -29782.984,E2 -29782.984} C_VEL
LIN {X 0,Y 189.894,Z 692.002,A -85,B 0,C 180,E1 -29787.709,E2 -29787.709} C_VEL
LIN {X 0,Y 198.964,Z 692.013,A -85,B 0,C 180,E1 -29790,E2 -29790} C_VEL
LIN {X 0,Y 189.895,Z 692.001,A -85,B 0,C 180,E1 -29792.292,E2 -29792.292} C_VEL
LIN {X 0,Y 172.632,Z 690.984,A -85,B 0,C 180,E1 -29797.015,E2 -29797.015} C_VEL
LIN {X 0,Y 158.143,Z 688.727,A -85,B 0,C 180,E1 -29802.146,E2 -29802.146} C_VEL
LIN {X 0,Y 147.211,Z 685.7,A -85,B 0,C 180,E1 -29807.305,E2 -29807.305} C_VEL
LIN {X 0,Y 137.826,Z 681.37,A -85,B 0,C 180,E1 -29813.399,E2 -29813.399} C_VEL
LIN {X 0,Y 131.877,Z 677.149,A -85,B 0,C 180,E1 -29818.661,E2 -29818.661} C_VEL
LIN {X 0,Y 127.346,Z 672.24,A -85,B 0,C 180,E1 -29824.134,E2 -29824.134} C_VEL
LIN {X 0,Y 123.758,Z 665.343,A -85,B 0,C 180,E1 -29830.784,E2 -29830.784} C_VEL
LIN {X 0,Y 122.156,Z 658.718,A -85,B 0,C 180,E1 -29836.346,E2 -29836.346} C_VEL
LIN {X 0,Y 121.626,Z 651.507,A -85,B 0,C 180,E1 -29841.606,E2 -29841.606} C_VEL
LIN {X 0,Y 122,Z 642.062,A -85,B 0,C 180,E1 -29847.418,E2 -29847.418} C_VEL
LIN {X 0,Y 122.909,Z 633.521,A -85,B 0,C 180,E1 -29851.882,E2 -29851.882} C_VEL
LIN {X 0,Y 124.24,Z 623.553,A -85,B 0,C 180,E1 -29856.237,E2 -29856.237} C_VEL
LIN {X 0,Y 125.349,Z 614.053,A -85,B 0,C 180,E1 -29859.933,E2 -29859.933} C_VEL
LIN {X 0,Y 125.448,Z 608.16,A -85,B 0,C 180,E1 -29862.817,E2 -29862.817} C_VEL
LIN {X 0,Y 124.953,Z 602.49,A -85,B 0,C 180,E1 -29866.383,E2 -29866.383} C_VEL
LIN {X 0,Y 124.37,Z 598.291,A -85,B 0,C 180,E1 -29870.245,E2 -29870.245} C_VEL
LIN {X 0,Y 123.824,Z 595.353,A -85,B 0,C 180,E1 -29874.305,E2 -29874.305} C_VEL
LIN {X 0,Y 123.694,Z 592.952,A -85,B 0,C 180,E1 -29880.005,E2 -29880.005} C_VEL
LIN {X 0,Y 124.01,Z 596.076,A -85,B 0,C 180,E1 -29886.513,E2 -29886.513} C_VEL
LIN {X 0,Y 124.567,Z 598.823,A -85,B 0,C 180,E1 -29889.862,E2 -29889.862} C_VEL
LIN {X 0,Y 121.455,Z 610.862,A -85,B 0,C 180,E1 -29890.361,E2 -29890.361} C_VEL
LIN {X 0,Y 117.672,Z 621.407,A -85,B 0,C 180,E1 -29890.872,E2 -29890.872} C_VEL
LIN {X 0,Y 112.984,Z 631.617,A -85,B 0,C 180,E1 -29891.566,E2 -29891.566} C_VEL
LIN {X 0,Y 107.926,Z 640.613,A -85,B 0,C 180,E1 -29892.374,E2 -29892.374} C_VEL
LIN {X 0,Y 102.054,Z 649.332,A -85,B 0,C 180,E1 -29893.415,E2 -29893.415} C_VEL
LIN {X 0,Y 96.235,Z 656.748,A -85,B 0,C 180,E1 -29894.618,E2 -29894.618} C_VEL
LIN {X 0,Y 88.016,Z 665.537,A -85,B 0,C 180,E1 -29896.628,E2 -29896.628} C_VEL
LIN {X 0,Y 81.542,Z 671.523,A -85,B 0,C 180,E1 -29898.546,E2 -29898.546} C_VEL
LIN {X 0,Y 73.629,Z 677.832,A -85,B 0,C 180,E1 -29901.465,E2 -29901.465} C_VEL
LIN {X 0,Y 65.787,Z 683.243,A -85,B 0,C 180,E1 -29905.307,E2 -29905.307} C_VEL
LIN {X 0,Y 57.262,Z 688.204,A -85,B 0,C 180,E1 -29910.781,E2 -29910.781} C_VEL
LIN {X 0,Y 49.203,Z 692.171,A -85,B 0,C 180,E1 -29918.225,E2 -29918.225} C_VEL
LIN {X 0,Y 42.252,Z 695.112,A -85,B 0,C 180,E1 -29928.292,E2 -29928.292} C_VEL
LIN {X 0,Y 38.629,Z 696.622,A -85,B 0,C 180,E1 -29936.921,E2 -29936.921} C_VEL
LIN {X 0,Y 34.427,Z 698.166,A -85,B 0,C 180,E1 -29958.221,E2 -29958.221} C_VEL
LIN {X 0,Y 34.18,Z 698.456,A -85,B 0,C 180,E1 -29970,E2 -29970} C_VEL
LIN {X 0,Y 35.974,Z 697.561,A -85,B 0,C 180,E1 -29993,E2 -29993} C_VEL
LIN {X 0,Y 38.63,Z 696.622,A -85,B 0,C 180,E1 -30003.079,E2 -30003.079} C_VEL
LIN {X 0,Y 46.734,Z 693.261,A -85,B 0,C 180,E1 -30018.756,E2 -30018.756} C_VEL
LIN {X 0,Y 54.455,Z 689.631,A -85,B 0,C 180,E1 -30027.023,E2 -30027.023} C_VEL
LIN {X 0,Y 60.131,Z 686.69,A -85,B 0,C 180,E1 -30031.233,E2 -30031.233} C_VEL
LIN {X 0,Y 69.013,Z 681.11,A -85,B 0,C 180,E1 -30036.421,E2 -30036.421} C_VEL
LIN {X 0,Y 76.771,Z 675.457,A -85,B 0,C 180,E1 -30039.773,E2 -30039.773} C_VEL
LIN {X 0,Y 84.769,Z 668.656,A -85,B 0,C 180,E1 -30042.444,E2 -30042.444} C_VEL
LIN {X 0,Y 92.924,Z 660.445,A -85,B 0,C 180,E1 -30044.643,E2 -30044.643} C_VEL
LIN {X 0,Y 99.554,Z 652.625,A -85,B 0,C 180,E1 -30046.088,E2 -30046.088} C_VEL
LIN {X 0,Y 105.413,Z 644.55,A -85,B 0,C 180,E1 -30047.176,E2 -30047.176} C_VEL
LIN {X 0,Y 111.29,Z 634.795,A -85,B 0,C 180,E1 -30048.186,E2 -30048.186} C_VEL
LIN {X 0,Y 115.855,Z 625.587,A -85,B 0,C 180,E1 -30048.911,E2 -30048.911} C_VEL
LIN {X 0,Y 119.767,Z 615.806,A -85,B 0,C 180,E1 -30049.478,E2 -30049.478} C_VEL
LIN {X 0,Y 123.075,Z 605.03,A -85,B 0,C 180,E1 -30049.861,E2 -30049.861} C_VEL
LIN {X 0,Y 124.57,Z 598.807,A -85,B 0,C 180,E1 -30050.138,E2 -30050.138} C_VEL
LIN {X 0,Y 123.892,Z 595.508,A -85,B 0,C 180,E1 -30054.298,E2 -30054.298} C_VEL
LIN {X 0,Y 123.652,Z 592.918,A -85,B 0,C 180,E1 -30060.402,E2 -30060.402} C_VEL
LIN {X 0,Y 123.927,Z 595.976,A -85,B 0,C 180,E1 -30066.712,E2 -30066.712} C_VEL
LIN {X 0,Y 124.448,Z 599.01,A -85,B 0,C 180,E1 -30070.468,E2 -30070.468} C_VEL
LIN {X 0,Y 124.999,Z 602.919,A -85,B 0,C 180,E1 -30073.923,E2 -30073.923} C_VEL
LIN {X 0,Y 125.457,Z 608.133,A -85,B 0,C 180,E1 -30077.181,E2 -30077.181} C_VEL
LIN {X 0,Y 125.35,Z 614.05,A -85,B 0,C 180,E1 -30080.067,E2 -30080.067} C_VEL
LIN {X 0,Y 124.387,Z 622.363,A -85,B 0,C 180,E1 -30083.292,E2 -30083.292} C_VEL
LIN {X 0,Y 123.326,Z 630.184,A -85,B 0,C 180,E1 -30086.579,E2 -30086.579} C_VEL
LIN {X 0,Y 122.354,Z 638.258,A -85,B 0,C 180,E1 -30090.504,E2 -30090.504} C_VEL
LIN {X 0,Y 121.693,Z 646.629,A -85,B 0,C 180,E1 -30095.27,E2 -30095.27} C_VEL
LIN {X 0,Y 121.708,Z 654.76,A -85,B 0,C 180,E1 -30100.69,E2 -30100.69} C_VEL
LIN {X 0,Y 122.815,Z 662.373,A -85,B 0,C 180,E1 -30106.632,E2 -30106.632} C_VEL
LIN {X 0,Y 124.983,Z 668.252,A -85,B 0,C 180,E1 -30111.92,E2 -30111.92} C_VEL
LIN {X 0,Y 128.763,Z 673.98,A -85,B 0,C 180,E1 -30117.766,E2 -30117.766} C_VEL
LIN {X 0,Y 133.824,Z 678.74,A -85,B 0,C 180,E1 -30123.213,E2 -30123.213} C_VEL
LIN {X 0,Y 142.332,Z 683.707,A -85,B 0,C 180,E1 -30129.779,E2 -30129.779} C_VEL
LIN {X 0,Y 146.941,Z 685.595,A -85,B 0,C 180,E1 -30132.546,E2 -30132.546} C_VEL
LIN {X 0,Y 149.788,Z 686.952,A -85,B 0,C 180,E1 -30134.481,E2 -30134.481} C_VEL
LIN {X 0,Y 155.018,Z 689.882,A -85,B 0,C 180,E1 -30139.191,E2 -30139.191} C_VEL
LIN {X 0,Y 158.92,Z 691.027,A -85,B 0,C 180,E1 -30141.654,E2 -30141.654} C_VEL
LIN {X 0,Y 161.506,Z 691.38,A -85,B 0,C 180,E1 -30142.701,E2 -30142.701} C_VEL
LIN {X 0,Y 178.802,Z 692.326,A -85,B 0,C 180,E1 -30147.747,E2 -30147.747} C_VEL
LIN {X 0,Y 187.844,Z 692.32,A -85,B 0,C 180,E1 -30150,E2 -30150} C_VEL
LIN {X 0,Y 175.927,Z 692.304,A -85,B 0,C 180,E1 -30152.997,E2 -30152.997} C_VEL
LIN {X 0,Y 160.822,Z 691.315,A -85,B 0,C 180,E1 -30157.533,E2 -30157.533} C_VEL
LIN {X 0,Y 150.569,Z 689.789,A -85,B 0,C 180,E1 -30161.445,E2 -30161.445} C_VEL
LIN {X 0,Y 138.23,Z 686.576,A -85,B 0,C 180,E1 -30167.761,E2 -30167.761} C_VEL
LIN {X 0,Y 128.309,Z 681.749,A -85,B 0,C 180,E1 -30175.159,E2 -30175.159} C_VEL
LIN {X 0,Y 122.856,Z 677.436,A -85,B 0,C 180,E1 -30180.987,E2 -30180.987} C_VEL
LIN {X 0,Y 118.556,Z 671.266,A -85,B 0,C 180,E1 -30188.141,E2 -30188.141} C_VEL
LIN {X 0,Y 116.679,Z 665.776,A -85,B 0,C 180,E1 -30193.722,E2 -30193.722} C_VEL
LIN {X 0,Y 115.855,Z 658.019,A -85,B 0,C 180,E1 -30200.445,E2 -30200.445} C_VEL
LIN {X 0,Y 116.315,Z 650.385,A -85,B 0,C 180,E1 -30206.027,E2 -30206.027} C_VEL
LIN {X 0,Y 117.329,Z 643.276,A -85,B 0,C 180,E1 -30210.516,E2 -30210.516} C_VEL
LIN {X 0,Y 119.164,Z 633.515,A -85,B 0,C 180,E1 -30215.623,E2 -30215.623} C_VEL
LIN {X 0,Y 120.994,Z 624.431,A -85,B 0,C 180,E1 -30219.609,E2 -30219.609} C_VEL
LIN {X 0,Y 122.306,Z 616.831,A -85,B 0,C 180,E1 -30222.791,E2 -30222.791} C_VEL
LIN {X 0,Y 122.553,Z 611.197,A -85,B 0,C 180,E1 -30225.899,E2 -30225.899} C_VEL
LIN {X 0,Y 122.538,Z 606.622,A -85,B 0,C 180,E1 -30229.366,E2 -30229.366} C_VEL
LIN {X 0,Y 122.222,Z 603.411,A -85,B 0,C 180,E1 -30232.987,E2 -30232.987} C_VEL
LIN {X 0,Y 122.109,Z 601.917,A -85,B 0,C 180,E1 -30235.466,E2 -30235.466} C_VEL
LIN {X 0,Y 122.264,Z 600.079,A -85,B 0,C 180,E1 -30240.005,E2 -30240.005} C_VEL
LIN {X 0,Y 122.275,Z 602.808,A -85,B 0,C 180,E1 -30245.778,E2 -30245.778} C_VEL
LIN {X 0,Y 122.327,Z 603.504,A -85,B 0,C 180,E1 -30246.706,E2 -30246.706} C_VEL
LIN {X 0,Y 120.38,Z 610.665,A -85,B 0,C 180,E1 -30247.03,E2 -30247.03} C_VEL
LIN {X 0,Y 116.225,Z 621.933,A -85,B 0,C 180,E1 -30247.477,E2 -30247.477} C_VEL
LIN {X 0,Y 111.777,Z 631.421,A -85,B 0,C 180,E1 -30247.999,E2 -30247.999} C_VEL
LIN {X 0,Y 106.63,Z 640.417,A -85,B 0,C 180,E1 -30248.644,E2 -30248.644} C_VEL
LIN {X 0,Y 100.646,Z 649.137,A -85,B 0,C 180,E1 -30249.486,E2 -30249.486} C_VEL
LIN {X 0,Y 94.693,Z 656.552,A -85,B 0,C 180,E1 -30250.458,E2 -30250.458} C_VEL
LIN {X 0,Y 86.249,Z 665.34,A -85,B 0,C 180,E1 -30252.093,E2 -30252.093} C_VEL
LIN {X 0,Y 79.56,Z 671.326,A -85,B 0,C 180,E1 -30253.668,E2 -30253.668} C_VEL
LIN {X 0,Y 71.326,Z 677.634,A -85,B 0,C 180,E1 -30256.117,E2 -30256.117} C_VEL
LIN {X 0,Y 62.234,Z 683.516,A -85,B 0,C 180,E1 -30259.813,E2 -30259.813} C_VEL
LIN {X 0,Y 53.969,Z 688.007,A -85,B 0,C 180,E1 -30264.28,E2 -30264.28} C_VEL
LIN {X 0,Y 45.142,Z 691.974,A -85,B 0,C 180,E1 -30271.1,E2 -30271.1} C_VEL
LIN {X 0,Y 37.228,Z 694.914,A -85,B 0,C 180,E1 -30280.963,E2 -30280.963} C_VEL
LIN {X 0,Y 32.893,Z 696.425,A -85,B 0,C 180,E1 -30290.135,E2 -30290.135} C_VEL
LIN {X 0,Y 27.507,Z 697.97,A -85,B 0,C 180,E1 -30315.197,E2 -30315.197} C_VEL
LIN {X 0,Y 27.07,Z 698.26,A -85,B 0,C 180,E1 -30330,E2 -30330} C_VEL
LIN {X 0,Y 29.536,Z 697.363,A -85,B 0,C 180,E1 -30358.417,E2 -30358.417} C_VEL
LIN {X 0,Y 32.893,Z 696.425,A -85,B 0,C 180,E1 -30369.865,E2 -30369.865} C_VEL
LIN {X 0,Y 42.373,Z 693.064,A -85,B 0,C 180,E1 -30386.026,E2 -30386.026} C_VEL
LIN {X 0,Y 50.93,Z 689.434,A -85,B 0,C 180,E1 -30393.76,E2 -30393.76} C_VEL
LIN {X 0,Y 60.143,Z 684.701,A -85,B 0,C 180,E1 -30399.199,E2 -30399.199} C_VEL
LIN {X 0,Y 69.708,Z 678.727,A -85,B 0,C 180,E1 -30403.292,E2 -30403.292} C_VEL
LIN {X 0,Y 77.911,Z 672.638,A -85,B 0,C 180,E1 -30405.858,E2 -30405.858} C_VEL
LIN {X 0,Y 84.57,Z 666.9,A -85,B 0,C 180,E1 -30407.539,E2 -30407.539} C_VEL
LIN {X 0,Y 91.299,Z 660.248,A -85,B 0,C 180,E1 -30408.949,E2 -30408.949} C_VEL
LIN {X 0,Y 98.088,Z 652.429,A -85,B 0,C 180,E1 -30410.121,E2 -30410.121} C_VEL
LIN {X 0,Y 104.066,Z 644.353,A -85,B 0,C 180,E1 -30410.996,E2 -30410.996} C_VEL
LIN {X 0,Y 110.058,Z 634.599,A -85,B 0,C 180,E1 -30411.801,E2 -30411.801} C_VEL
LIN {X 0,Y 115.047,Z 624.593,A -85,B 0,C 180,E1 -30412.443,E2 -30412.443} C_VEL
LIN {X 0,Y 118.909,Z 614.923,A -85,B 0,C 180,E1 -30412.877,E2 -30412.877} C_VEL
LIN {X 0,Y 121.959,Z 605.104,A -85,B 0,C 180,E1 -30413.133,E2 -30413.133} C_VEL
LIN {X 0,Y 122.33,Z 603.511,A -85,B 0,C 180,E1 -30413.276,E2 -30413.276} C_VEL
LIN {X 0,Y 122.183,Z 601.881,A -85,B 0,C 180,E1 -30415.872,E2 -30415.872} C_VEL
LIN {X 0,Y 122.265,Z 600.064,A -85,B 0,C 180,E1 -30420.407,E2 -30420.407} C_VEL
LIN {X 0,Y 122.185,Z 602.812,A -85,B 0,C 180,E1 -30426.186,E2 -30426.186} C_VEL
LIN {X 0,Y 122.484,Z 606.08,A -85,B 0,C 180,E1 -30430.116,E2 -30430.116} C_VEL
LIN {X 0,Y 122.596,Z 609.498,A -85,B 0,C 180,E1 -30432.957,E2 -30432.957} C_VEL
LIN {X 0,Y 122.481,Z 614.009,A -85,B 0,C 180,E1 -30435.811,E2 -30435.811} C_VEL
LIN {X 0,Y 121.935,Z 619.295,A -85,B 0,C 180,E1 -30438.318,E2 -30438.318} C_VEL
LIN {X 0,Y 120.051,Z 629.122,A -85,B 0,C 180,E1 -30442.358,E2 -30442.358} C_VEL
LIN {X 0,Y 118.179,Z 638.498,A -85,B 0,C 180,E1 -30446.871,E2 -30446.871} C_VEL
LIN {X 0,Y 116.754,Z 646.836,A -85,B 0,C 180,E1 -30451.65,E2 -30451.65} C_VEL
LIN {X 0,Y 115.914,Z 655.114,A -85,B 0,C 180,E1 -30457.316,E2 -30457.316} C_VEL
LIN {X 0,Y 116.145,Z 662.634,A -85,B 0,C 180,E1 -30463.438,E2 -30463.438} C_VEL
LIN {X 0,Y 117.364,Z 668.366,A -85,B 0,C 180,E1 -30468.799,E2 -30468.799} C_VEL
LIN {X 0,Y 120.214,Z 674.02,A -85,B 0,C 180,E1 -30474.922,E2 -30474.922} C_VEL
LIN {X 0,Y 124.544,Z 678.99,A -85,B 0,C 180,E1 -30480.993,E2 -30480.993} C_VEL
LIN {X 0,Y 132.216,Z 684.002,A -85,B 0,C 180,E1 -30488.156,E2 -30488.156} C_VEL
LIN {X 0,Y 141.221,Z 687.5,A -85,B 0,C 180,E1 -30494.001,E2 -30494.001} C_VEL
LIN {X 0,Y 152.509,Z 690.108,A -85,B 0,C 180,E1 -30499.378,E2 -30499.378} C_VEL
LIN {X 0,Y 161.506,Z 691.38,A -85,B 0,C 180,E1 -30502.701,E2 -30502.701} C_VEL
LIN {X 0,Y 163.907,Z 691.729,A -85,B 0,C 180,E1 -30503.813,E2 -30503.813} C_VEL
LIN {X 0,Y 166.592,Z 692.356,A -85,B 0,C 180,E1 -30505.949,E2 -30505.949} C_VEL
LIN {X 0,Y 169.504,Z 692.629,A -85,B 0,C 180,E1 -30508.016,E2 -30508.016} C_VEL
LIN {X 0,Y 172.183,Z 692.656,A -85,B 0,C 180,E1 -30509.001,E2 -30509.001} C_VEL
LIN {X 0,Y 176.225,Z 692.641,A -85,B 0,C 180,E1 -30510,E2 -30510} C_VEL
LIN {X 0,Y 157.763,Z 692.317,A -85,B 0,C 180,E1 -30515.112,E2 -30515.112} C_VEL
LIN {X 0,Y 149.086,Z 691.63,A -85,B 0,C 180,E1 -30518.164,E2 -30518.164} C_VEL
LIN {X 0,Y 137.293,Z 689.679,A -85,B 0,C 180,E1 -30523.464,E2 -30523.464} C_VEL
LIN {X 0,Y 127.028,Z 686.518,A -85,B 0,C 180,E1 -30529.873,E2 -30529.873} C_VEL
LIN {X 0,Y 118.766,Z 681.957,A -85,B 0,C 180,E1 -30537.436,E2 -30537.436} C_VEL
LIN {X 0,Y 114.33,Z 677.715,A -85,B 0,C 180,E1 -30543.589,E2 -30543.589} C_VEL
LIN {X 0,Y 111.23,Z 672.021,A -85,B 0,C 180,E1 -30550.702,E2 -30550.702} C_VEL
LIN {X 0,Y 109.977,Z 665.26,A -85,B 0,C 180,E1 -30557.867,E2 -30557.867} C_VEL
LIN {X 0,Y 110.255,Z 658.182,A -85,B 0,C 180,E1 -30564.193,E2 -30564.193} C_VEL
LIN {X 0,Y 111.546,Z 650.769,A -85,B 0,C 180,E1 -30569.739,E2 -30569.739} C_VEL
LIN {X 0,Y 113.522,Z 642.497,A -85,B 0,C 180,E1 -30574.939,E2 -30574.939} C_VEL
LIN {X 0,Y 116.207,Z 632.612,A -85,B 0,C 180,E1 -30579.979,E2 -30579.979} C_VEL
LIN {X 0,Y 118.468,Z 624.097,A -85,B 0,C 180,E1 -30583.639,E2 -30583.639} C_VEL
LIN {X 0,Y 119.281,Z 620.139,A -85,B 0,C 180,E1 -30585.504,E2 -30585.504} C_VEL
LIN {X 0,Y 119.815,Z 616.365,A -85,B 0,C 180,E1 -30587.786,E2 -30587.786} C_VEL
LIN {X 0,Y 119.999,Z 613.523,A -85,B 0,C 180,E1 -30589.886,E2 -30589.886} C_VEL
LIN {X 0,Y 120.136,Z 610.336,A -85,B 0,C 180,E1 -30593.286,E2 -30593.286} C_VEL
LIN {X 0,Y 120.251,Z 608.398,A -85,B 0,C 180,E1 -30596.655,E2 -30596.655} C_VEL
LIN {X 0,Y 120.471,Z 607.102,A -85,B 0,C 180,E1 -30600.005,E2 -30600.005} C_VEL
LIN {X 0,Y 120.322,Z 608.563,A -85,B 0,C 180,E1 -30603.354,E2 -30603.354} C_VEL
LIN {X 0,Y 119.718,Z 610.469,A -85,B 0,C 180,E1 -30603.653,E2 -30603.653} C_VEL
LIN {X 0,Y 115.518,Z 621.735,A -85,B 0,C 180,E1 -30603.989,E2 -30603.989} C_VEL
LIN {X 0,Y 111.012,Z 631.225,A -85,B 0,C 180,E1 -30604.37,E2 -30604.37} C_VEL
LIN {X 0,Y 105.795,Z 640.22,A -85,B 0,C 180,E1 -30604.835,E2 -30604.835} C_VEL
LIN {X 0,Y 99.722,Z 648.94,A -85,B 0,C 180,E1 -30605.462,E2 -30605.462} C_VEL
LIN {X 0,Y 93.665,Z 656.356,A -85,B 0,C 180,E1 -30606.185,E2 -30606.185} C_VEL
LIN {X 0,Y 85.045,Z 665.144,A -85,B 0,C 180,E1 -30607.408,E2 -30607.408} C_VEL
LIN {X 0,Y 78.185,Z 671.129,A -85,B 0,C 180,E1 -30608.596,E2 -30608.596} C_VEL
LIN {X 0,Y 69.685,Z 677.437,A -85,B 0,C 180,E1 -30610.482,E2 -30610.482} C_VEL
LIN {X 0,Y 61.304,Z 682.715,A -85,B 0,C 180,E1 -30612.995,E2 -30612.995} C_VEL
LIN {X 0,Y 51.453,Z 687.81,A -85,B 0,C 180,E1 -30617.037,E2 -30617.037} C_VEL
LIN {X 0,Y 41.907,Z 691.777,A -85,B 0,C 180,E1 -30622.727,E2 -30622.727} C_VEL
LIN {X 0,Y 32.992,Z 694.717,A -85,B 0,C 180,E1 -30631.562,E2 -30631.562} C_VEL
LIN {X 0,Y 27.794,Z 696.228,A -85,B 0,C 180,E1 -30640.662,E2 -30640.662} C_VEL
LIN {X 0,Y 20.701,Z 697.773,A -85,B 0,C 180,E1 -30670.154,E2 -30670.154} C_VEL
LIN {X 0,Y 19.976,Z 698.064,A -85,B 0,C 180,E1 -30690,E2 -30690} C_VEL
LIN {X 0,Y 23.515,Z 697.166,A -85,B 0,C 180,E1 -30726.707,E2 -30726.707} C_VEL
LIN {X 0,Y 27.795,Z 696.228,A -85,B 0,C 180,E1 -30739.337,E2 -30739.337} C_VEL
LIN {X 0,Y 38.843,Z 692.867,A -85,B 0,C 180,E1 -30754.777,E2 -30754.777} C_VEL
LIN {X 0,Y 48.208,Z 689.237,A -85,B 0,C 180,E1 -30761.369,E2 -30761.369} C_VEL
LIN {X 0,Y 58,Z 684.505,A -85,B 0,C 180,E1 -30765.783,E2 -30765.783} C_VEL
LIN {X 0,Y 66.32,Z 679.623,A -85,B 0,C 180,E1 -30768.584,E2 -30768.584} C_VEL
LIN {X 0,Y 74.777,Z 673.752,A -85,B 0,C 180,E1 -30770.695,E2 -30770.695} C_VEL
LIN {X 0,Y 81.611,Z 668.263,A -85,B 0,C 180,E1 -30772.02,E2 -30772.02} C_VEL
LIN {X 0,Y 90.204,Z 660.051,A -85,B 0,C 180,E1 -30773.398,E2 -30773.398} C_VEL
LIN {X 0,Y 97.123,Z 652.232,A -85,B 0,C 180,E1 -30774.25,E2 -30774.25} C_VEL
LIN {X 0,Y 103.193,Z 644.157,A -85,B 0,C 180,E1 -30774.893,E2 -30774.893} C_VEL
LIN {X 0,Y 109.271,Z 634.402,A -85,B 0,C 180,E1 -30775.489,E2 -30775.489} C_VEL
LIN {X 0,Y 113.591,Z 626.073,A -85,B 0,C 180,E1 -30775.899,E2 -30775.899} C_VEL
LIN {X 0,Y 117.791,Z 616.027,A -85,B 0,C 180,E1 -30776.251,E2 -30776.251} C_VEL
LIN {X 0,Y 119.713,Z 610.467,A -85,B 0,C 180,E1 -30776.382,E2 -30776.382} C_VEL
LIN {X 0,Y 120.335,Z 608.521,A -85,B 0,C 180,E1 -30776.647,E2 -30776.647} C_VEL
LIN {X 0,Y 120.469,Z 607.11,A -85,B 0,C 180,E1 -30779.995,E2 -30779.995} C_VEL
LIN {X 0,Y 120.253,Z 608.39,A -85,B 0,C 180,E1 -30783.345,E2 -30783.345} C_VEL
LIN {X 0,Y 120.127,Z 610.362,A -85,B 0,C 180,E1 -30786.714,E2 -30786.714} C_VEL
LIN {X 0,Y 119.997,Z 613.529,A -85,B 0,C 180,E1 -30790.114,E2 -30790.114} C_VEL
LIN {X 0,Y 119.57,Z 618.538,A -85,B 0,C 180,E1 -30793.593,E2 -30793.593} C_VEL
LIN {X 0,Y 118.482,Z 624.063,A -85,B 0,C 180,E1 -30796.359,E2 -30796.359} C_VEL
LIN {X 0,Y 115.472,Z 635.581,A -85,B 0,C 180,E1 -30801.413,E2 -30801.413} C_VEL
LIN {X 0,Y 112.455,Z 646.761,A -85,B 0,C 180,E1 -30807.607,E2 -30807.607} C_VEL
LIN {X 0,Y 110.579,Z 655.613,A -85,B 0,C 180,E1 -30813.749,E2 -30813.749} C_VEL
LIN {X 0,Y 109.935,Z 662.712,A -85,B 0,C 180,E1 -30819.731,E2 -30819.731} C_VEL
LIN {X 0,Y 110.315,Z 668.631,A -85,B 0,C 180,E1 -30825.51,E2 -30825.51} C_VEL
LIN {X 0,Y 112.154,Z 674.284,A -85,B 0,C 180,E1 -30831.963,E2 -30831.963} C_VEL
LIN {X 0,Y 116.674,Z 680.215,A -85,B 0,C 180,E1 -30839.961,E2 -30839.961} C_VEL
LIN {X 0,Y 122.619,Z 684.395,A -85,B 0,C 180,E1 -30846.484,E2 -30846.484} C_VEL
LIN {X 0,Y 127.858,Z 686.878,A -85,B 0,C 180,E1 -30850.743,E2 -30850.743} C_VEL
LIN {X 0,Y 137.289,Z 689.685,A -85,B 0,C 180,E1 -30856.543,E2 -30856.543} C_VEL
LIN {X 0,Y 149.161,Z 691.643,A -85,B 0,C 180,E1 -30861.874,E2 -30861.874} C_VEL
LIN {X 0,Y 161.987,Z 692.582,A -85,B 0,C 180,E1 -30866.199,E2 -30866.199} C_VEL
LIN {X 0,Y 172.183,Z 692.656,A -85,B 0,C 180,E1 -30869.001,E2 -30869.001} C_VEL
LIN {X 0,Y 170.718,Z 692.729,A -85,B 0,C 180,E1 -30869.109,E2 -30869.109} C_VEL
LIN {X 0,Y 164.095,Z 692.826,A -85,B 0,C 180,E1 -30868.398,E2 -30868.398} C_VEL
LIN {X 0,Y 153.607,Z 692.903,A -85,B 0,C 180,E1 -30866.461,E2 -30866.461} C_VEL
LIN {X 0,Y 146.357,Z 692.655,A -85,B 0,C 180,E1 -30864.557,E2 -30864.557} C_VEL
LIN {X 0,Y 144.157,Z 692.496,A -85,B 0,C 180,E1 -30863.795,E2 -30863.795} C_VEL
LIN {X 0,Y 135.499,Z 691.643,A -85,B 0,C 180,E1 -30860.195,E2 -30860.195} C_VEL
LIN {X 0,Y 123.553,Z 689.136,A -85,B 0,C 180,E1 -30853.476,E2 -30853.476} C_VEL
LIN {X 0,Y 117.835,Z 687.173,A -85,B 0,C 180,E1 -30849.032,E2 -30849.032} C_VEL
LIN {X 0,Y 111.274,Z 683.514,A -85,B 0,C 180,E1 -30842.143,E2 -30842.143} C_VEL
LIN {X 0,Y 105.892,Z 677.522,A -85,B 0,C 180,E1 -30832.78,E2 -30832.78} C_VEL
LIN {X 0,Y 103.973,Z 671.759,A -85,B 0,C 180,E1 -30825.185,E2 -30825.185} C_VEL
LIN {X 0,Y 103.867,Z 666.196,A -85,B 0,C 180,E1 -30818.962,E2 -30818.962} C_VEL
LIN {X 0,Y 105.005,Z 659.171,A -85,B 0,C 180,E1 -30812.366,E2 -30812.366} C_VEL
LIN {X 0,Y 107.436,Z 650.711,A -85,B 0,C 180,E1 -30805.96,E2 -30805.96} C_VEL
LIN {X 0,Y 109.83,Z 643.76,A -85,B 0,C 180,E1 -30801.581,E2 -30801.581} C_VEL
LIN {X 0,Y 113.097,Z 634.38,A -85,B 0,C 180,E1 -30796.719,E2 -30796.719} C_VEL
LIN {X 0,Y 115.908,Z 625.867,A -85,B 0,C 180,E1 -30792.925,E2 -30792.925} C_VEL
LIN {X 0,Y 116.838,Z 621.638,A -85,B 0,C 180,E1 -30790.391,E2 -30790.391} C_VEL
